C05497=1155.282,-127.548,-42.199,178.609,5.885,149.463
C05498=1155.288,-127.798,-42.191,178.606,5.885,149.464
C05499=1155.293,-128.048,-42.183,178.605,5.885,149.465
C05500=1154.872,-128.059,-42.224,178.601,5.888,149.466
C05501=1154.867,-127.809,-42.233,178.603,5.888,149.466
C05502=1154.861,-127.559,-42.241,178.605,5.888,149.465
C05503=1154.855,-127.309,-42.250,178.607,5.889,149.465
C05504=1154.850,-127.060,-42.259,178.609,5.889,149.464
C05505=1154.845,-126.809,-42.267,178.611,5.890,149.464
C05506=1154.840,-126.560,-42.275,178.613,5.890,149.463
C05507=1154.834,-126.310,-42.283,178.615,5.890,149.463
C05508=1154.829,-126.060,-42.292,178.617,5.890,149.462
C05509=1154.823,-125.811,-42.301,178.619,5.891,149.462
C05510=1154.818,-125.560,-42.309,178.621,5.891,149.461
C05511=1154.813,-125.311,-42.318,178.623,5.891,149.461
C05512=1154.807,-125.061,-42.326,178.624,5.891,149.460
C05513=1154.802,-124.811,-42.334,178.627,5.892,149.460
C05514=1154.797,-124.561,-42.343,178.628,5.892,149.459
C05515=1154.791,-124.312,-42.351,178.631,5.892,149.458
C05516=1154.786,-124.062,-42.359,178.632,5.892,149.458
C05517=1154.781,-123.812,-42.368,178.635,5.893,149.457
C05518=1154.775,-123.563,-42.377,178.636,5.893,149.457
C05519=1154.769,-123.312,-42.385,178.638,5.894,149.457
C05520=1154.764,-123.062,-42.394,178.640,5.894,149.456
C05521=1154.758,-122.813,-42.402,178.642,5.895,149.456
C05522=1154.753,-122.563,-42.411,178.644,5.894,149.455
C05523=1154.749,-122.313,-42.419,178.647,5.895,149.454
C05524=1154.743,-122.064,-42.427,178.648,5.895,149.454
C05525=1154.738,-121.814,-42.436,178.650,5.896,149.453
C05526=1154.732,-121.564,-42.445,178.652,5.896,149.453
C05527=1154.727,-121.314,-42.453,178.654,5.896,149.452
C05528=1154.721,-121.065,-42.462,178.657,5.897,149.452
C05529=1154.716,-120.815,-42.471,178.658,5.897,149.451
C05530=1154.711,-120.564,-42.479,178.661,5.897,149.451
C05531=1154.705,-120.315,-42.488,178.662,5.897,149.450
C05532=1154.700,-120.065,-42.496,178.664,5.898,149.450
C05533=1154.694,-119.816,-42.505,178.666,5.898,149.449
C05534=1154.689,-119.565,-42.514,178.669,5.898,149.449
C05535=1154.683,-119.316,-42.522,178.670,5.898,149.448
C05536=1154.678,-119.066,-42.531,178.672,5.899,149.448
C05537=1154.673,-118.816,-42.540,178.674,5.899,149.447
C05538=1154.668,-118.566,-42.549,178.676,5.900,149.447
C05539=1154.662,-118.317,-42.557,178.678,5.899,149.446
C05540=1154.656,-118.067,-42.565,178.681,5.900,149.445
C05541=1154.651,-117.817,-42.574,178.682,5.900,149.445
C05542=1154.646,-117.567,-42.583,178.684,5.901,149.444
C05543=1154.640,-117.318,-42.592,178.686,5.901,149.444
C05544=1154.635,-117.068,-42.601,178.689,5.901,149.443
C05545=1154.630,-116.818,-42.609,178.691,5.902,149.443
C05546=1154.625,-116.568,-42.618,178.692,5.902,149.442
C05547=1154.619,-116.318,-42.627,178.695,5.903,149.442
C05548=1154.614,-116.069,-42.635,178.696,5.903,149.441
C05549=1154.608,-115.819,-42.644,178.698,5.903,149.441
C05550=1154.603,-115.569,-42.653,178.700,5.903,149.440
C05551=1154.598,-115.319,-42.662,178.703,5.904,149.440
C05552=1154.592,-115.070,-42.670,178.704,5.904,149.439
C05553=1154.587,-114.820,-42.679,178.706,5.904,149.439
C05554=1154.582,-114.570,-42.688,178.708,5.904,149.438
C05555=1154.577,-114.320,-42.696,178.711,5.905,149.437
C05556=1154.571,-114.070,-42.705,178.712,5.905,149.437
C05557=1154.566,-113.821,-42.714,178.715,5.906,149.436
C05558=1154.560,-113.571,-42.723,178.717,5.906,149.436
C05559=1154.555,-113.321,-42.732,178.719,5.906,149.435
C05560=1154.549,-113.071,-42.741,178.721,5.907,149.435
C05561=1154.544,-112.821,-42.750,178.723,5.907,149.434
C05562=1154.539,-112.571,-42.759,178.725,5.907,149.434
C05563=1154.533,-112.322,-42.767,178.726,5.907,149.433
C05564=1154.528,-112.072,-42.776,178.729,5.908,149.433
C05565=1154.523,-111.822,-42.785,178.731,5.908,149.432
C05566=1154.518,-111.573,-42.794,178.733,5.908,149.432
C05567=1154.512,-111.322,-42.804,178.735,5.909,149.431
C05568=1154.507,-111.073,-42.813,178.737,5.909,149.431
C05569=1154.501,-110.823,-42.821,178.739,5.909,149.430
C05570=1154.496,-110.574,-42.830,178.741,5.909,149.429
C05571=1154.491,-110.324,-42.839,178.743,5.910,149.429
C05572=1154.485,-110.074,-42.848,178.745,5.910,149.428
C05573=1154.480,-109.824,-42.857,178.747,5.911,149.428
C05574=1154.474,-109.574,-42.866,178.750,5.911,149.427
C05575=1154.469,-109.324,-42.875,178.751,5.911,149.427
C05576=1154.463,-109.075,-42.884,178.753,5.912,149.426
C05577=1154.458,-108.825,-42.893,178.755,5.912,149.426
C05578=1154.453,-108.575,-42.901,178.758,5.912,149.425
C05579=1154.448,-108.325,-42.910,178.759,5.912,149.425
C05580=1154.442,-108.075,-42.920,178.761,5.913,149.424
C05581=1154.437,-107.825,-42.929,178.764,5.914,149.424
C05582=1154.432,-107.575,-42.938,178.766,5.913,149.423
C05583=1154.427,-107.326,-42.947,178.768,5.914,149.422
C05584=1154.421,-107.077,-42.956,178.770,5.914,149.422
C05585=1154.415,-106.827,-42.965,178.772,5.915,149.421
C05586=1154.410,-106.577,-42.974,178.774,5.914,149.421
C05587=1154.405,-106.327,-42.983,178.776,5.915,149.420
C05588=1154.400,-106.077,-42.992,178.778,5.916,149.420
C05589=1154.395,-105.828,-43.001,178.780,5.916,149.419
C05590=1154.389,-105.577,-43.010,178.782,5.916,149.419
C05591=1154.383,-105.328,-43.019,178.784,5.916,149.418
C05592=1154.379,-105.078,-43.029,178.786,5.917,149.418
C05593=1154.373,-104.828,-43.038,178.788,5.917,149.417
C05594=1154.368,-104.578,-43.047,178.791,5.917,149.416
C05595=1154.362,-104.328,-43.056,178.793,5.918,149.416
C05596=1154.357,-104.079,-43.065,178.794,5.918,149.415
C05597=1154.351,-103.829,-43.074,178.797,5.919,149.415
C05598=1154.346,-103.580,-43.084,178.799,5.918,149.414
C05599=1154.341,-103.330,-43.093,178.801,5.919,149.414
C05600=1154.335,-103.080,-43.102,178.803,5.920,149.413
C05601=1154.330,-102.808,-43.112,178.805,5.920,149.413
C05602=1154.324,-102.536,-43.121,178.807,5.920,149.412
C05603=1154.318,-102.263,-43.132,178.810,5.921,149.411
C05604=1154.312,-101.992,-43.142,178.812,5.921,149.411
C05605=1154.307,-101.742,-43.151,178.814,5.921,149.410
C05606=1154.302,-101.492,-43.160,178.816,5.922,149.410
C05607=1154.296,-101.243,-43.170,178.818,5.922,149.409
C05608=1154.291,-100.993,-43.179,178.820,5.922,149.409
C05609=1154.286,-100.743,-43.188,178.822,5.923,149.408
C05610=1154.280,-100.493,-43.197,178.824,5.923,149.407
C05611=1154.275,-100.244,-43.207,178.827,5.924,149.407
C05612=1154.270,-99.994,-43.216,178.828,5.924,149.407
C05613=1154.264,-99.744,-43.225,178.830,5.924,149.406
C05614=1154.259,-99.495,-43.235,178.833,5.925,149.405
C05615=1154.254,-99.245,-43.244,178.835,5.925,149.405
C05616=1154.248,-98.995,-43.253,178.837,5.925,149.404
C05617=1154.243,-98.745,-43.262,178.839,5.925,149.404
C05618=1154.238,-98.496,-43.272,178.841,5.926,149.403
C05619=1154.232,-98.245,-43.281,178.843,5.927,149.403
C05620=1154.227,-97.996,-43.290,178.845,5.927,149.402
C05621=1154.221,-97.746,-43.300,178.848,5.927,149.401
C05622=1154.216,-97.496,-43.309,178.850,5.928,149.401
C05623=1154.211,-97.246,-43.318,178.851,5.928,149.400
C05624=1154.205,-96.997,-43.328,178.854,5.928,149.400
C05625=1154.200,-96.747,-43.337,178.856,5.928,149.399
C05626=1154.194,-96.497,-43.348,178.858,5.929,149.399
C05627=1154.189,-96.248,-43.356,178.860,5.929,149.398
C05628=1154.185,-95.997,-43.366,178.862,5.929,149.398
C05629=1154.179,-95.747,-43.376,178.864,5.930,149.397
C05630=1154.174,-95.498,-43.385,178.867,5.931,149.397
C05631=1154.168,-95.248,-43.395,178.869,5.930,149.396
C05632=1154.163,-94.998,-43.404,178.871,5.931,149.395
C05633=1154.157,-94.748,-43.413,178.872,5.931,149.395
C05634=1154.152,-94.499,-43.423,178.875,5.932,149.394
C05635=1154.147,-94.249,-43.432,178.877,5.932,149.394
C05636=1154.142,-93.999,-43.442,178.879,5.932,149.393
C05637=1154.136,-93.750,-43.451,178.881,5.933,149.393
C05638=1154.131,-93.500,-43.461,178.884,5.933,149.392
C05639=1154.126,-93.250,-43.470,178.885,5.933,149.392
C05640=1154.120,-93.001,-43.480,178.888,5.934,149.391
C05641=1154.115,-92.751,-43.489,178.890,5.934,149.390
C05642=1154.109,-92.501,-43.499,178.892,5.934,149.390
C05643=1154.104,-92.251,-43.508,178.894,5.935,149.389
C05644=1154.099,-92.001,-43.519,178.896,5.935,149.389
C05645=1154.094,-91.751,-43.528,178.898,5.935,149.388
C05646=1154.088,-91.502,-43.538,178.900,5.936,149.388
C05647=1154.083,-91.252,-43.547,178.902,5.936,149.387
C05648=1154.078,-91.002,-43.557,178.905,5.936,149.387
C05649=1154.072,-90.752,-43.566,178.907,5.937,149.386
C05650=1154.067,-90.503,-43.576,178.909,5.937,149.386
C05651=1154.062,-90.253,-43.585,178.911,5.938,149.385
C05652=1154.056,-90.004,-43.595,178.913,5.938,149.384
C05653=1154.052,-89.753,-43.605,178.915,5.938,149.384
C05654=1154.046,-89.503,-43.615,178.918,5.939,149.383
C05655=1154.041,-89.254,-43.624,178.920,5.939,149.383
C05656=1154.035,-89.004,-43.634,178.921,5.939,149.382
C05657=1154.030,-88.755,-43.644,178.924,5.940,149.382
C05658=1154.024,-88.505,-43.653,178.926,5.941,149.381
C05659=1154.019,-88.255,-43.663,178.928,5.941,149.381
C05660=1154.014,-88.005,-43.672,178.931,5.941,149.380
C05661=1154.009,-87.755,-43.683,178.933,5.942,149.379
C05662=1154.004,-87.506,-43.692,178.934,5.942,149.379
C05663=1153.998,-87.256,-43.702,178.937,5.942,149.378
C05664=1153.992,-87.006,-43.712,178.939,5.943,149.378
C05665=1153.987,-86.757,-43.722,178.941,5.943,149.377
C05666=1153.982,-86.507,-43.731,178.943,5.944,149.377
C05667=1153.977,-86.257,-43.741,178.946,5.944,149.376
C05668=1153.972,-86.007,-43.751,178.947,5.944,149.376
C05669=1153.966,-85.757,-43.761,178.949,5.945,149.375
C05670=1153.961,-85.508,-43.770,178.952,5.945,149.374
C05671=1153.955,-85.258,-43.781,178.954,5.945,149.374
C05672=1153.951,-85.008,-43.790,178.956,5.946,149.373
C05673=1153.945,-84.758,-43.800,178.959,5.946,149.373
C05674=1153.940,-84.509,-43.810,178.960,5.946,149.372
C05675=1153.934,-84.259,-43.819,178.962,5.947,149.372
C05676=1153.929,-84.009,-43.829,178.965,5.947,149.371
C05677=1153.924,-83.759,-43.840,178.967,5.947,149.371
C05678=1153.919,-83.510,-43.850,178.969,5.948,149.370
C05679=1153.913,-83.260,-43.859,178.972,5.948,149.369
C05680=1153.907,-83.010,-43.869,178.973,5.948,149.369
C05681=1153.903,-82.761,-43.879,178.976,5.949,149.368
C05682=1153.898,-82.511,-43.889,178.978,5.950,149.368
C05683=1153.892,-82.260,-43.899,178.980,5.950,149.367
C05684=1153.887,-82.011,-43.909,178.982,5.950,149.366
C05685=1153.881,-81.762,-43.919,178.984,5.951,149.366
C05686=1153.876,-81.511,-43.929,178.986,5.951,149.365
C05687=1153.871,-81.262,-43.938,178.989,5.951,149.365
C05688=1153.865,-81.012,-43.948,178.991,5.952,149.364
C05689=1153.860,-80.762,-43.959,178.993,5.953,149.364
C05690=1153.854,-80.513,-43.969,178.995,5.952,149.363
C05691=1153.850,-80.263,-43.979,178.997,5.953,149.363
C05692=1153.844,-80.013,-43.989,179.000,5.954,149.362
C05693=1153.838,-79.763,-43.999,179.002,5.953,149.361
C05694=1153.834,-79.513,-44.009,179.004,5.954,149.361
C05695=1153.829,-79.264,-44.019,179.006,5.955,149.360
C05696=1153.823,-79.014,-44.029,179.008,5.954,149.360
C05697=1153.817,-78.765,-44.039,179.010,5.955,149.359
C05698=1153.812,-78.514,-44.050,179.013,5.956,149.359
C05699=1153.808,-78.265,-44.059,179.015,5.956,149.358
C05700=1153.802,-78.015,-44.069,179.017,5.956,149.358
C05701=1153.796,-77.766,-44.079,179.019,5.957,149.357
C05702=1153.791,-77.515,-44.090,179.022,5.958,149.356
C05703=1153.786,-77.266,-44.099,179.023,5.958,149.356
C05704=1153.781,-77.017,-44.109,179.026,5.958,149.355
C05705=1153.775,-76.745,-44.121,179.028,5.959,149.355
C05706=1153.770,-76.474,-44.132,179.031,5.959,149.354
C05707=1153.763,-76.203,-44.143,179.033,5.960,149.354
C05708=1153.758,-75.931,-44.154,179.036,5.960,149.353
C05709=1153.752,-75.681,-44.164,179.037,5.960,149.352
C05710=1153.747,-75.431,-44.174,179.040,5.961,149.352
C05711=1153.741,-75.181,-44.184,179.042,5.961,149.351
C05712=1153.736,-74.932,-44.195,179.044,5.961,149.351
C05713=1153.731,-74.682,-44.205,179.046,5.962,149.350
C05714=1153.726,-74.432,-44.215,179.049,5.963,149.349
C05715=1153.720,-74.183,-44.225,179.051,5.963,149.349
C05716=1153.715,-73.933,-44.235,179.053,5.963,149.348
C05717=1153.710,-73.683,-44.246,179.055,5.964,149.348
C05718=1153.704,-73.434,-44.256,179.058,5.964,149.347
C05719=1153.698,-73.184,-44.266,179.060,5.965,149.347
C05720=1153.694,-72.934,-44.276,179.061,5.965,149.346
C05721=1153.689,-72.685,-44.286,179.064,5.965,149.345
C05722=1153.684,-72.434,-44.297,179.066,5.966,149.345
C05723=1153.678,-72.185,-44.308,179.069,5.966,149.344
C05724=1153.673,-71.936,-44.318,179.071,5.966,149.344
C05725=1153.668,-71.686,-44.329,179.073,5.967,149.343
C05726=1153.662,-71.436,-44.339,179.075,5.967,149.343
C05727=1153.657,-71.186,-44.349,179.077,5.967,149.342
C05728=1153.652,-70.936,-44.360,179.079,5.968,149.342
C05729=1153.646,-70.687,-44.370,179.082,5.969,149.341
C05730=1153.640,-70.437,-44.380,179.084,5.969,149.340
C05731=1153.635,-70.187,-44.391,179.086,5.969,149.340
C05732=1153.630,-69.938,-44.400,179.088,5.970,149.339
C05733=1153.625,-69.687,-44.411,179.091,5.971,149.339
C05734=1153.620,-69.438,-44.421,179.093,5.971,149.338
C05735=1153.615,-69.189,-44.432,179.095,5.971,149.338
C05736=1153.610,-68.939,-44.442,179.097,5.971,149.337
C05737=1153.604,-68.689,-44.453,179.100,5.972,149.336
C05738=1153.599,-68.439,-44.463,179.102,5.973,149.336
C05739=1153.593,-68.189,-44.473,179.104,5.972,149.335
C05740=1153.588,-67.940,-44.484,179.106,5.973,149.335
C05741=1153.583,-67.690,-44.495,179.109,5.974,149.334
C05742=1153.577,-67.441,-44.505,179.111,5.974,149.334
C05743=1153.572,-67.190,-44.516,179.113,5.974,149.333
C05744=1153.567,-66.941,-44.526,179.115,5.975,149.332
C05745=1153.562,-66.691,-44.537,179.117,5.976,149.332
C05746=1153.557,-66.442,-44.547,179.120,5.976,149.331
C05747=1153.552,-66.191,-44.558,179.122,5.977,149.331
C05748=1153.546,-65.942,-44.568,179.124,5.977,149.330
C05749=1153.540,-65.692,-44.578,179.127,5.977,149.329
C05750=1153.536,-65.443,-44.590,179.129,5.978,149.329
C05751=1153.530,-65.193,-44.600,179.131,5.979,149.329
C05752=1153.525,-64.943,-44.611,179.133,5.978,149.328
C05753=1153.520,-64.693,-44.621,179.135,5.979,149.327
C05754=1153.515,-64.444,-44.632,179.138,5.979,149.327
C05755=1153.509,-64.194,-44.642,179.140,5.980,149.326
C05756=1153.504,-63.944,-44.653,179.142,5.981,149.326
C05757=1153.498,-63.694,-44.664,179.144,5.981,149.325
C05758=1153.493,-63.445,-44.675,179.146,5.981,149.324
C05759=1153.488,-63.195,-44.685,179.149,5.982,149.324
C05760=1153.483,-62.945,-44.696,179.151,5.983,149.323
C05761=1153.477,-62.696,-44.707,179.153,5.982,149.323
C05762=1153.472,-62.446,-44.717,179.156,5.983,149.322
C05763=1153.467,-62.196,-44.727,179.158,5.984,149.322
C05764=1153.462,-61.946,-44.739,179.160,5.984,149.321
C05765=1153.456,-61.697,-44.749,179.163,5.985,149.320
C05766=1153.451,-61.447,-44.759,179.165,5.984,149.320
C05767=1153.446,-61.198,-44.770,179.167,5.985,149.319
C05768=1153.440,-60.947,-44.782,179.169,5.986,149.319
C05769=1153.435,-60.698,-44.792,179.172,5.986,149.318
C05770=1153.430,-60.448,-44.803,179.174,5.987,149.318
C05771=1153.425,-60.198,-44.813,179.176,5.987,149.317
C05772=1153.420,-59.949,-44.825,179.178,5.988,149.316
C05773=1153.414,-59.699,-44.835,179.180,5.988,149.316
C05774=1153.410,-59.450,-44.846,179.183,5.989,149.315
C05775=1153.404,-59.200,-44.856,179.185,5.990,149.315
C05776=1153.398,-58.950,-44.867,179.187,5.989,149.314
C05777=1153.394,-58.700,-44.879,179.190,5.990,149.314
C05778=1153.388,-58.450,-44.889,179.192,5.990,149.313
C05779=1153.383,-58.201,-44.900,179.194,5.991,149.312
C05780=1153.378,-57.951,-44.910,179.197,5.992,149.312
C05781=1153.373,-57.702,-44.922,179.199,5.992,149.311
C05782=1153.367,-57.452,-44.933,179.201,5.992,149.311
C05783=1153.362,-57.202,-44.944,179.204,5.993,149.310
C05784=1153.357,-56.952,-44.954,179.206,5.993,149.310
C05785=1153.352,-56.703,-44.965,179.208,5.994,149.309
C05786=1153.347,-56.453,-44.976,179.210,5.994,149.308
C05787=1153.341,-56.203,-44.987,179.212,5.995,149.308
C05788=1153.336,-55.953,-44.998,179.215,5.995,149.307
C05789=1153.331,-55.704,-45.009,179.217,5.996,149.307
C05790=1153.325,-55.454,-45.019,179.220,5.996,149.306
C05791=1153.320,-55.204,-45.031,179.222,5.997,149.306
C05792=1153.314,-54.955,-45.042,179.223,5.997,149.305
C05793=1153.310,-54.705,-45.053,179.226,5.997,149.304
C05794=1153.305,-54.455,-45.063,179.228,5.998,149.304
C05795=1153.299,-54.205,-45.075,179.231,5.999,149.303
C05796=1153.294,-53.956,-45.086,179.233,5.999,149.303
C05797=1153.288,-53.706,-45.096,179.235,5.999,149.302
C05798=1153.284,-53.457,-45.108,179.237,6.000,149.301
C05799=1153.278,-53.206,-45.119,179.240,6.001,149.301
C05800=1153.273,-52.957,-45.130,179.242,6.001,149.300
C05801=1153.268,-52.708,-45.141,179.244,6.002,149.300
C05802=1153.262,-52.457,-45.152,179.247,6.002,149.299
C05803=1153.257,-52.208,-45.163,179.249,6.002,149.299
C05804=1153.252,-51.958,-45.175,179.251,6.003,149.298
C05805=1153.247,-51.708,-45.185,179.254,6.003,149.297
C05806=1153.241,-51.459,-45.197,179.256,6.004,149.297
C05807=1153.236,-51.209,-45.208,179.258,6.005,149.296
C05808=1153.231,-50.959,-45.218,179.261,6.005,149.296
C05809=1153.225,-50.689,-45.230,179.263,6.006,149.295
C05810=1153.220,-50.418,-45.243,179.266,6.006,149.294
C05811=1153.214,-50.148,-45.255,179.268,6.007,149.294
C05812=1153.208,-49.877,-45.267,179.271,6.007,149.293
C05813=1153.203,-49.627,-45.278,179.273,6.008,149.293
C05814=1153.197,-49.378,-45.290,179.275,6.008,149.292
C05815=1153.192,-49.128,-45.301,179.277,6.008,149.292
C05816=1153.187,-48.878,-45.311,179.280,6.009,149.291
C05817=1153.182,-48.628,-45.323,179.282,6.010,149.290
C05818=1153.177,-48.379,-45.334,179.285,6.010,149.290
C05819=1153.172,-48.129,-45.346,179.287,6.011,149.289
C05820=1153.166,-47.879,-45.357,179.289,6.012,149.289
C05821=1153.161,-47.630,-45.368,179.291,6.011,149.288
C05822=1153.155,-47.380,-45.379,179.293,6.012,149.288
C05823=1153.151,-47.130,-45.391,179.296,6.012,149.287
C05824=1153.145,-46.881,-45.402,179.298,6.013,149.286
C05825=1153.140,-46.631,-45.413,179.301,6.014,149.286
C05826=1153.135,-46.381,-45.424,179.303,6.014,149.285
C05827=1153.130,-46.131,-45.436,179.306,6.015,149.284
C05828=1153.124,-45.882,-45.447,179.307,6.015,149.284
C05829=1153.119,-45.632,-45.459,179.310,6.016,149.284
C05830=1153.114,-45.383,-45.470,179.312,6.016,149.283
C05831=1153.108,-45.132,-45.481,179.314,6.017,149.282
C05832=1153.103,-44.883,-45.492,179.317,6.017,149.282
C05833=1153.098,-44.633,-45.504,179.319,6.018,149.281
C05834=1153.093,-44.384,-45.515,179.322,6.018,149.280
C05835=1153.088,-44.134,-45.527,179.324,6.019,149.280
C05836=1153.082,-43.885,-45.538,179.327,6.020,149.279
C05837=1153.077,-43.635,-45.550,179.328,6.020,149.279
C05838=1153.072,-43.385,-45.561,179.331,6.020,149.278
C05839=1153.066,-43.135,-45.573,179.333,6.021,149.278
C05840=1153.061,-42.886,-45.583,179.335,6.022,149.277
C05841=1153.056,-42.636,-45.595,179.338,6.022,149.276
C05842=1153.051,-42.386,-45.607,179.340,6.023,149.276
C05843=1153.046,-42.136,-45.619,179.343,6.023,149.275
C05844=1153.041,-41.887,-45.630,179.345,6.024,149.275
C05845=1153.035,-41.637,-45.641,179.348,6.024,149.274
C05846=1153.030,-41.388,-45.653,179.349,6.024,149.274
C05847=1153.025,-41.138,-45.665,179.352,6.025,149.273
C05848=1153.020,-40.888,-45.676,179.354,6.026,149.272
C05849=1153.015,-40.638,-45.688,179.356,6.026,149.272
C05850=1153.010,-40.389,-45.699,179.359,6.027,149.271
C05851=1153.004,-40.140,-45.711,179.361,6.028,149.271
C05852=1152.999,-39.890,-45.722,179.364,6.028,149.270
C05853=1152.994,-39.640,-45.734,179.366,6.029,149.270
C05854=1152.988,-39.390,-45.746,179.369,6.029,149.269
C05855=1152.984,-39.140,-45.757,179.371,6.030,149.268
C05856=1152.978,-38.891,-45.768,179.373,6.030,149.268
C05857=1152.972,-38.641,-45.780,179.375,6.030,149.267
C05858=1152.968,-38.392,-45.792,179.378,6.031,149.267
C05859=1152.962,-38.142,-45.803,179.380,6.032,149.266
C05860=1152.957,-37.892,-45.815,179.382,6.032,149.266
C05861=1152.952,-37.642,-45.827,179.385,6.033,149.265
C05862=1152.947,-37.392,-45.839,179.387,6.034,149.264
C05863=1152.942,-37.144,-45.850,179.390,6.034,149.264
C05864=1152.936,-36.894,-45.862,179.392,6.035,149.263
C05865=1152.931,-36.644,-45.874,179.395,6.035,149.263
C05866=1152.926,-36.394,-45.885,179.397,6.036,149.262
C05867=1152.921,-36.144,-45.897,179.399,6.036,149.261
C05868=1152.915,-35.894,-45.909,179.401,6.036,149.261
C05869=1152.910,-35.645,-45.920,179.404,6.037,149.260
C05870=1152.905,-35.395,-45.932,179.406,6.038,149.260
C05871=1152.899,-35.146,-45.944,179.409,6.038,149.259
C05872=1152.895,-34.897,-45.956,179.411,6.039,149.259
C05873=1152.889,-34.647,-45.968,179.413,6.040,149.258
C05874=1152.884,-34.397,-45.979,179.416,6.040,149.257
C05875=1152.878,-34.147,-45.991,179.418,6.041,149.257
C05876=1152.874,-33.897,-46.003,179.420,6.041,149.256
C05877=1152.869,-33.648,-46.015,179.423,6.042,149.256
C05878=1152.863,-33.398,-46.027,179.425,6.042,149.255
C05879=1152.858,-33.148,-46.038,179.427,6.043,149.255
C05880=1152.853,-32.898,-46.050,179.430,6.044,149.254
C05881=1152.848,-32.648,-46.062,179.432,6.044,149.253
C05882=1152.842,-32.399,-46.075,179.435,6.045,149.253
C05883=1152.837,-32.150,-46.086,179.437,6.046,149.252
C05884=1152.832,-31.900,-46.098,179.439,6.045,149.252
C05885=1152.827,-31.651,-46.110,179.441,6.046,149.251
C05886=1152.821,-31.401,-46.122,179.444,6.047,149.250
C05887=1152.816,-31.151,-46.133,179.446,6.047,149.250
C05888=1152.811,-30.901,-46.145,179.448,6.048,149.249
C05889=1152.806,-30.652,-46.158,179.451,6.049,149.249
C05890=1152.800,-30.402,-46.170,179.453,6.049,149.248
C05891=1152.795,-30.152,-46.182,179.456,6.050,149.248
C05892=1152.791,-29.903,-46.194,179.458,6.051,149.247
C05893=1152.785,-29.653,-46.206,179.461,6.051,149.246
C05894=1152.780,-29.403,-46.217,179.463,6.052,149.246
C05895=1152.775,-29.154,-46.230,179.466,6.052,149.245
C05896=1152.769,-28.904,-46.242,179.468,6.053,149.245
C05897=1152.765,-28.655,-46.253,179.470,6.053,149.244
C05898=1152.759,-28.405,-46.266,179.473,6.054,149.244
C05899=1152.754,-28.155,-46.278,179.475,6.055,149.243
C05900=1152.749,-27.905,-46.290,179.477,6.055,149.242
C05901=1152.743,-27.656,-46.302,179.480,6.056,149.242
C05902=1152.738,-27.406,-46.314,179.482,6.057,149.241
C05903=1152.734,-27.157,-46.326,179.485,6.057,149.241
C05904=1152.728,-26.907,-46.338,179.487,6.058,149.240
C05905=1152.723,-26.657,-46.350,179.489,6.059,149.240
C05906=1152.718,-26.408,-46.362,179.492,6.059,149.239
C05907=1152.712,-26.158,-46.374,179.494,6.060,149.238
C05908=1152.707,-25.909,-46.387,179.497,6.060,149.238
C05909=1152.702,-25.659,-46.399,179.499,6.061,149.237
C05910=1152.697,-25.409,-46.411,179.502,6.062,149.237
C05911=1152.691,-25.159,-46.423,179.504,6.062,149.236
C05912=1152.687,-24.910,-46.435,179.507,6.063,149.235
C05913=1152.681,-24.640,-46.449,179.509,6.064,149.235
C05914=1152.675,-24.369,-46.462,179.511,6.064,149.234
C05915=1152.670,-24.100,-46.475,179.514,6.064,149.234
C05916=1152.664,-23.830,-46.488,179.517,6.065,149.233
C05917=1152.659,-23.581,-46.501,179.519,6.066,149.232
C05918=1152.654,-23.331,-46.513,179.521,6.066,149.232
C05919=1152.649,-23.081,-46.525,179.524,6.067,149.231
C05920=1152.643,-22.832,-46.537,179.526,6.068,149.231
C05921=1152.638,-22.582,-46.550,179.529,6.068,149.230
C05922=1152.633,-22.332,-46.562,179.531,6.069,149.230
C05923=1152.628,-22.082,-46.574,179.533,6.069,149.229
C05924=1152.623,-21.832,-46.586,179.536,6.070,149.228
C05925=1152.618,-21.583,-46.599,179.538,6.071,149.228
C05926=1152.613,-21.334,-46.612,179.540,6.071,149.227
C05927=1152.607,-21.084,-46.623,179.543,6.072,149.227
C05928=1152.602,-20.834,-46.636,179.545,6.073,149.226
C05929=1152.597,-20.585,-46.648,179.548,6.073,149.225
C05930=1152.592,-20.335,-46.661,179.550,6.074,149.225
C05931=1152.586,-20.086,-46.673,179.553,6.074,149.224
C05932=1152.582,-19.835,-46.685,179.555,6.075,149.224
C05933=1152.576,-19.586,-46.698,179.558,6.075,149.223
C05934=1152.571,-19.337,-46.711,179.560,6.076,149.223
C05935=1152.566,-19.087,-46.722,179.562,6.077,149.222
C05936=1152.561,-18.837,-46.735,179.565,6.077,149.221
C05937=1152.555,-18.588,-46.748,179.567,6.078,149.221
C05938=1152.549,-18.338,-46.760,179.569,6.079,149.220
C05939=1152.545,-18.088,-46.773,179.572,6.080,149.220
C05940=1152.540,-17.838,-46.786,179.575,6.081,149.219
C05941=1152.534,-17.588,-46.798,179.577,6.082,149.219
C05942=1152.529,-17.339,-46.810,179.580,6.082,149.218
C05943=1152.524,-17.090,-46.823,179.582,6.083,149.217
C05944=1152.519,-16.841,-46.835,179.585,6.083,149.217
C05945=1152.514,-16.590,-46.848,179.587,6.084,149.216
C05946=1152.509,-16.341,-46.860,179.589,6.084,149.216
C05947=1152.504,-16.091,-46.873,179.592,6.085,149.215
C05948=1152.498,-15.842,-46.886,179.594,6.086,149.214
C05949=1152.493,-15.592,-46.898,179.596,6.086,149.214
C05950=1152.488,-15.342,-46.911,179.599,6.087,149.213
C05951=1152.483,-15.092,-46.924,179.601,6.088,149.213
C05952=1152.478,-14.843,-46.936,179.604,6.088,149.212
C05953=1152.473,-14.594,-46.949,179.606,6.089,149.212
C05954=1152.468,-14.344,-46.961,179.609,6.089,149.211
C05955=1152.462,-14.093,-46.974,179.611,6.090,149.210
C05956=1152.457,-13.844,-46.987,179.614,6.091,149.210
C05957=1152.452,-13.595,-46.999,179.616,6.091,149.209
C05958=1152.447,-13.346,-47.012,179.618,6.092,149.209
C05959=1152.442,-13.096,-47.025,179.621,6.093,149.208
C05960=1152.437,-12.846,-47.038,179.623,6.093,149.207
C05961=1152.431,-12.596,-47.050,179.625,6.094,149.207
C05962=1152.426,-12.347,-47.063,179.629,6.095,149.206
C05963=1152.421,-12.097,-47.075,179.631,6.096,149.206
C05964=1152.416,-11.847,-47.088,179.634,6.096,149.205
C05965=1152.411,-11.598,-47.101,179.636,6.097,149.205
C05966=1152.405,-11.348,-47.114,179.638,6.098,149.204
C05967=1152.400,-11.099,-47.127,179.641,6.098,149.203
C05968=1152.395,-10.849,-47.140,179.643,6.099,149.203
C05969=1152.390,-10.600,-47.152,179.645,6.100,149.202
C05970=1152.384,-10.350,-47.165,179.648,6.100,149.202
C05971=1152.380,-10.100,-47.178,179.650,6.101,149.201
C05972=1152.375,-9.851,-47.191,179.652,6.102,149.201
C05973=1152.370,-9.601,-47.204,179.655,6.102,149.200
C05974=1152.364,-9.352,-47.217,179.657,6.103,149.200
C05975=1152.359,-9.102,-47.230,179.660,6.103,149.199
C05976=1152.354,-8.852,-47.242,179.663,6.105,149.198
C05977=1152.348,-8.603,-47.255,179.665,6.105,149.198
C05978=1152.344,-8.353,-47.268,179.668,6.106,149.197
C05979=1152.339,-8.103,-47.281,179.670,6.107,149.197
C05980=1152.334,-7.854,-47.294,179.672,6.107,149.196
C05981=1152.328,-7.604,-47.307,179.675,6.108,149.195
C05982=1152.323,-7.355,-47.320,179.677,6.109,149.195
C05983=1152.318,-7.105,-47.332,179.680,6.109,149.194
C05984=1152.313,-6.855,-47.346,179.682,6.110,149.194
C05985=1152.308,-6.606,-47.359,179.685,6.110,149.193
C05986=1152.303,-6.356,-47.371,179.687,6.111,149.193
C05987=1152.297,-6.106,-47.385,179.690,6.112,149.192
C05988=1152.292,-5.857,-47.397,179.692,6.113,149.191
C05989=1152.287,-5.608,-47.411,179.695,6.114,149.191
C05990=1152.282,-5.358,-47.424,179.697,6.114,149.190
C05991=1152.277,-5.108,-47.437,179.700,6.115,149.190
C05992=1152.271,-4.859,-47.450,179.702,6.116,149.189
C05993=1152.267,-4.609,-47.463,179.705,6.116,149.188
C05994=1152.261,-4.359,-47.476,179.707,6.117,149.188
C05995=1152.256,-4.109,-47.489,179.709,6.118,149.188
C05996=1152.251,-3.860,-47.502,179.712,6.119,149.187
C05997=1152.246,-3.611,-47.516,179.714,6.120,149.186
C05998=1152.241,-3.361,-47.529,179.717,6.120,149.186
C05999=1152.236,-3.111,-47.541,179.719,6.121,149.185
C06000=1152.231,-2.861,-47.555,179.722,6.122,149.185
C06001=1152.226,-2.612,-47.568,179.724,6.122,149.184
C06002=1152.220,-2.363,-47.581,179.727,6.123,149.183
C06003=1152.215,-2.113,-47.594,179.729,6.124,149.183
C06004=1152.210,-1.863,-47.607,179.732,6.124,149.182
C06005=1152.205,-1.614,-47.621,179.734,6.126,149.182
C06006=1152.199,-1.364,-47.634,179.737,6.126,149.181
C06007=1152.194,-1.115,-47.647,179.739,6.127,149.181
C06008=1152.190,-0.865,-47.660,179.742,6.127,149.180
C06009=1152.184,-0.616,-47.674,179.744,6.128,149.179
C06010=1152.180,-0.366,-47.687,179.747,6.129,149.179
C06011=1152.174,-0.116,-47.700,179.749,6.129,149.178
C06012=1152.169,0.134,-47.713,179.752,6.131,149.178
C06013=1152.164,0.383,-47.727,179.754,6.131,149.177
C06014=1152.159,0.632,-47.739,179.757,6.132,149.176
C06015=1152.153,0.883,-47.753,179.759,6.133,149.176
C06016=1152.148,1.132,-47.767,179.762,6.133,149.175
C06017=1152.143,1.401,-47.781,179.764,6.134,149.175
C06018=1152.137,1.671,-47.796,179.767,6.135,149.174
C06019=1152.132,1.941,-47.810,179.770,6.136,149.173
C06020=1152.126,2.209,-47.824,179.772,6.136,149.173
C06021=1152.121,2.460,-47.837,179.775,6.138,149.172
C06022=1152.116,2.709,-47.851,179.777,6.139,149.172
C06023=1152.111,2.959,-47.864,179.780,6.139,149.171
C06024=1152.106,3.208,-47.878,179.782,6.140,149.171
C06025=1152.101,3.458,-47.891,179.785,6.140,149.170
C06026=1152.095,3.707,-47.904,179.787,6.141,149.170
C06027=1152.091,3.957,-47.918,179.790,6.142,149.169
C06028=1152.085,4.206,-47.931,179.792,6.143,149.168
C06029=1152.080,4.456,-47.946,179.795,6.144,149.168
C06030=1152.075,4.705,-47.958,179.797,6.144,149.167
C06031=1152.070,4.955,-47.972,179.800,6.145,149.167
C06032=1152.065,5.204,-47.985,179.802,6.146,149.166
C06033=1152.060,5.454,-47.999,179.805,6.146,149.165
C06034=1152.054,5.704,-48.013,179.808,6.148,149.165
C06035=1152.050,5.953,-48.026,179.810,6.148,149.164
C06036=1152.044,6.203,-48.039,179.812,6.149,149.164
C06037=1152.039,6.452,-48.054,179.815,6.150,149.163
C06038=1152.035,6.703,-48.067,179.817,6.150,149.163
C06039=1152.029,6.952,-48.081,179.820,6.152,149.162
C06040=1152.024,7.202,-48.094,179.823,6.152,149.161
C06041=1152.019,7.451,-48.107,179.825,6.153,149.161
C06042=1152.014,7.700,-48.122,179.827,6.154,149.160
C06043=1152.008,7.950,-48.135,179.830,6.154,149.160
C06044=1152.004,8.199,-48.149,179.832,6.155,149.159
C06045=1151.999,8.450,-48.162,179.835,6.156,149.159
C06046=1151.993,8.699,-48.176,179.838,6.157,149.158
C06047=1151.989,8.948,-48.190,179.840,6.158,149.158
C06048=1151.983,9.198,-48.203,179.843,6.158,149.157
C06049=1151.978,9.447,-48.217,179.845,6.159,149.156
C06050=1151.973,9.698,-48.231,179.848,6.160,149.156
C06051=1151.968,9.946,-48.244,179.850,6.161,149.155
C06052=1151.963,10.196,-48.258,179.853,6.162,149.155
C06053=1151.957,10.446,-48.272,179.855,6.162,149.154
C06054=1151.952,10.695,-48.286,179.858,6.163,149.153
C06055=1151.948,10.945,-48.300,179.860,6.164,149.153
C06056=1151.942,11.194,-48.313,179.863,6.165,149.152
C06057=1151.937,11.444,-48.327,179.865,6.166,149.152
C06058=1151.932,11.693,-48.341,179.867,6.167,149.151
C06059=1151.927,11.943,-48.355,179.870,6.167,149.151
C06060=1151.922,12.193,-48.368,179.873,6.169,149.150
C06061=1151.917,12.442,-48.382,179.875,6.169,149.150
C06062=1151.912,12.692,-48.396,179.878,6.170,149.149
C06063=1151.906,12.942,-48.410,179.880,6.170,149.148
C06064=1151.901,13.191,-48.424,179.882,6.171,149.148
C06065=1151.897,13.440,-48.438,179.886,6.172,149.147
C06066=1151.892,13.690,-48.452,179.888,6.173,149.147
C06067=1151.886,13.939,-48.466,179.890,6.174,149.146
C06068=1151.881,14.189,-48.479,179.893,6.174,149.146
C06069=1151.876,14.439,-48.494,179.896,6.176,149.145
C06070=1151.870,14.688,-48.507,179.898,6.177,149.145
C06071=1151.866,14.938,-48.521,179.901,6.177,149.144
C06072=1151.861,15.187,-48.535,179.903,6.178,149.143
C06073=1151.855,15.437,-48.549,179.906,6.179,149.143
C06074=1151.850,15.687,-48.563,179.908,6.180,149.142
C06075=1151.845,15.936,-48.577,179.910,6.181,149.142
C06076=1151.840,16.186,-48.591,179.913,6.181,149.141
C06077=1151.835,16.435,-48.605,179.915,6.182,149.141
C06078=1151.830,16.685,-48.620,179.919,6.183,149.140
C06079=1151.825,16.934,-48.634,179.921,6.184,149.140
C06080=1151.819,17.183,-48.648,179.923,6.185,149.139
C06081=1151.815,17.433,-48.661,179.926,6.185,149.138
C06082=1151.810,17.683,-48.675,179.929,6.187,149.138
C06083=1151.805,17.933,-48.689,179.931,6.187,149.137
C06084=1151.799,18.182,-48.703,179.934,6.188,149.137
C06085=1151.794,18.432,-48.718,179.936,6.189,149.136
C06086=1151.789,18.681,-48.732,179.939,6.190,149.135
C06087=1151.784,18.931,-48.746,179.941,6.191,149.135
C06088=1151.779,19.180,-48.760,179.944,6.191,149.134
C06089=1151.774,19.430,-48.774,179.946,6.192,149.134
C06090=1151.769,19.679,-48.789,179.949,6.193,149.133
C06091=1151.764,19.929,-48.803,179.951,6.194,149.133
C06092=1151.758,20.178,-48.817,179.954,6.195,149.132
C06093=1151.754,20.428,-48.831,179.957,6.196,149.132
C06094=1151.749,20.678,-48.845,179.959,6.197,149.131
C06095=1151.744,20.927,-48.860,179.962,6.198,149.130
C06096=1151.739,21.177,-48.874,179.964,6.198,149.130
C06097=1151.733,21.426,-48.888,179.967,6.200,149.129
C06098=1151.728,21.676,-48.902,179.969,6.200,149.129
C06099=1151.723,21.925,-48.916,179.972,6.201,149.128
C06100=1151.718,22.175,-48.931,179.974,6.202,149.128
C06101=1151.714,22.424,-48.946,179.977,6.203,149.127
C06102=1151.708,22.673,-48.959,179.979,6.204,149.127
C06103=1151.703,22.923,-48.974,179.982,6.204,149.126
C06104=1151.698,23.173,-48.988,179.985,6.206,149.125
C06105=1151.693,23.422,-49.002,179.987,6.207,149.125
C06106=1151.687,23.672,-49.017,179.990,6.207,149.124
C06107=1151.683,23.922,-49.031,179.992,6.208,149.124
C06108=1151.677,24.171,-49.045,179.995,6.209,149.123
C06109=1151.672,24.420,-49.060,179.997,6.210,149.123
C06110=1151.667,24.670,-49.075,180.000,6.211,149.122
C06111=1151.662,24.920,-49.089,-179.997,6.212,149.122
C06112=1151.657,25.169,-49.103,-179.995,6.213,149.121
C06113=1151.653,25.419,-49.117,-179.993,6.214,149.120
C06114=1151.647,25.668,-49.131,-179.990,6.214,149.120
C06115=1151.642,25.917,-49.147,-179.987,6.216,149.119
C06116=1151.637,26.167,-49.161,-179.984,6.216,149.119
C06117=1151.632,26.417,-49.176,-179.982,6.217,149.118
C06118=1151.627,26.667,-49.190,-179.980,6.219,149.118
C06119=1151.622,26.916,-49.205,-179.977,6.219,149.117
C06120=1151.617,27.165,-49.219,-179.975,6.220,149.117
C06121=1151.611,27.435,-49.235,-179.971,6.221,149.116
C06122=1151.606,27.704,-49.250,-179.969,6.222,149.115
C06123=1151.600,27.972,-49.266,-179.966,6.223,149.115
C06124=1151.595,28.241,-49.281,-179.963,6.224,149.114
C06125=1151.589,28.491,-49.296,-179.961,6.225,149.114
C06126=1151.585,28.740,-49.311,-179.958,6.226,149.113
C06127=1151.580,28.990,-49.326,-179.956,6.227,149.112
C06128=1151.575,29.239,-49.340,-179.953,6.228,149.112
C06129=1151.569,29.489,-49.355,-179.950,6.229,149.111
C06130=1151.564,29.738,-49.370,-179.948,6.229,149.111
C06131=1151.559,29.988,-49.384,-179.946,6.230,149.110
C06132=1151.555,30.237,-49.399,-179.942,6.231,149.110
C06133=1151.550,30.487,-49.413,-179.940,6.232,149.109
C06134=1151.544,30.736,-49.429,-179.938,6.233,149.109
C06135=1151.539,30.986,-49.443,-179.935,6.234,149.108
C06136=1151.535,31.236,-49.457,-179.933,6.235,149.108
C06137=1151.529,31.485,-49.473,-179.930,6.235,149.107
C06138=1151.524,31.735,-49.487,-179.927,6.237,149.106
C06139=1151.520,31.984,-49.502,-179.925,6.238,149.106
C06140=1151.514,32.233,-49.516,-179.922,6.238,149.105
C06141=1151.509,32.482,-49.532,-179.919,6.240,149.105
C06142=1151.504,32.732,-49.546,-179.917,6.241,149.104
C06143=1151.499,32.982,-49.560,-179.914,6.242,149.104
C06144=1151.493,33.231,-49.576,-179.912,6.243,149.103
C06145=1151.488,33.481,-49.590,-179.909,6.243,149.103
C06146=1151.484,33.730,-49.605,-179.906,6.245,149.102
C06147=1151.478,33.980,-49.620,-179.904,6.246,149.101
C06148=1151.473,34.229,-49.635,-179.901,6.246,149.101
C06149=1151.468,34.479,-49.649,-179.899,6.248,149.100
C06150=1151.463,34.728,-49.665,-179.896,6.248,149.100
C06151=1151.459,34.978,-49.680,-179.894,6.249,149.099
C06152=1151.453,35.228,-49.695,-179.891,6.251,149.099
C06153=1151.449,35.477,-49.710,-179.888,6.251,149.098
C06154=1151.444,35.727,-49.724,-179.886,6.252,149.098
C06155=1151.438,35.976,-49.740,-179.883,6.253,149.097
C06156=1151.433,36.226,-49.754,-179.881,6.254,149.096
C06157=1151.428,36.475,-49.770,-179.878,6.255,149.096
C06158=1151.423,36.724,-49.785,-179.875,6.256,149.095
C06159=1151.418,36.974,-49.799,-179.873,6.257,149.095
C06160=1151.413,37.224,-49.815,-179.870,6.258,149.094
C06161=1151.408,37.473,-49.829,-179.868,6.259,149.094
C06162=1151.403,37.723,-49.845,-179.865,6.260,149.093
C06163=1151.398,37.972,-49.860,-179.863,6.261,149.093
C06164=1151.392,38.222,-49.874,-179.860,6.262,149.092
C06165=1151.388,38.471,-49.889,-179.857,6.263,149.092
C06166=1151.382,38.720,-49.905,-179.854,6.264,149.091
C06167=1151.377,38.970,-49.919,-179.852,6.265,149.090
C06168=1151.373,39.219,-49.934,-179.850,6.266,149.090
C06169=1151.368,39.469,-49.950,-179.847,6.267,149.089
C06170=1151.363,39.718,-49.965,-179.845,6.268,149.089
C06171=1151.357,39.968,-49.980,-179.842,6.269,149.088
C06172=1151.353,40.217,-49.995,-179.839,6.270,149.088
C06173=1151.347,40.467,-50.011,-179.836,6.271,149.087
C06174=1151.342,40.716,-50.026,-179.834,6.272,149.087
C06175=1151.337,40.966,-50.041,-179.832,6.273,149.086
C06176=1151.332,41.215,-50.056,-179.829,6.274,149.085
C06177=1151.328,41.465,-50.071,-179.826,6.275,149.085
C06178=1151.322,41.715,-50.087,-179.823,6.276,149.084
C06179=1151.317,41.964,-50.101,-179.821,6.277,149.084
C06180=1151.312,42.214,-50.117,-179.818,6.277,149.083
C06181=1151.307,42.463,-50.132,-179.816,6.279,149.083
C06182=1151.302,42.712,-50.148,-179.813,6.280,149.082
C06183=1151.297,42.961,-50.163,-179.810,6.281,149.082
C06184=1151.292,43.211,-50.178,-179.808,6.282,149.081
C06185=1151.287,43.461,-50.193,-179.805,6.283,149.081
C06186=1151.282,43.710,-50.208,-179.803,6.284,149.080
C06187=1151.277,43.960,-50.224,-179.800,6.285,149.079
C06188=1151.272,44.209,-50.239,-179.797,6.286,149.079
C06189=1151.267,44.458,-50.255,-179.795,6.287,149.079
C06190=1151.262,44.708,-50.270,-179.792,6.288,149.078
C06191=1151.257,44.958,-50.285,-179.790,6.289,149.077
C06192=1151.252,45.207,-50.301,-179.786,6.290,149.077
C06193=1151.246,45.456,-50.317,-179.784,6.291,149.076
C06194=1151.242,45.706,-50.332,-179.782,6.292,149.076
C06195=1151.237,45.956,-50.348,-179.779,6.293,149.075
C06196=1151.232,46.205,-50.363,-179.777,6.294,149.075
C06197=1151.227,46.454,-50.378,-179.774,6.296,149.074
C06198=1151.222,46.703,-50.394,-179.771,6.296,149.074
C06199=1151.217,46.954,-50.410,-179.768,6.298,149.073
C06200=1151.212,47.203,-50.425,-179.766,6.299,149.073
C06201=1151.207,47.452,-50.440,-179.764,6.299,149.072
C06202=1151.201,47.701,-50.456,-179.761,6.301,149.071
C06203=1151.197,47.951,-50.471,-179.758,6.302,149.071
C06204=1151.192,48.201,-50.487,-179.755,6.303,149.070
C06205=1151.187,48.450,-50.502,-179.753,6.304,149.070
C06206=1151.182,48.699,-50.517,-179.750,6.305,149.069
C06207=1151.177,48.949,-50.533,-179.748,6.306,149.069
C06208=1151.172,49.199,-50.549,-179.745,6.307,149.068
C06209=1151.166,49.448,-50.565,-179.742,6.308,149.068
C06210=1151.162,49.697,-50.580,-179.740,6.309,149.067
C06211=1151.157,49.947,-50.595,-179.737,6.310,149.067
C06212=1151.152,50.197,-50.611,-179.735,6.311,149.066
C06213=1151.146,50.446,-50.627,-179.732,6.313,149.066
C06214=1151.142,50.695,-50.643,-179.729,6.313,149.065
C06215=1151.137,50.945,-50.658,-179.727,6.315,149.065
C06216=1151.132,51.194,-50.674,-179.724,6.316,149.064
C06217=1151.127,51.444,-50.690,-179.721,6.317,149.063
C06218=1151.121,51.694,-50.705,-179.719,6.318,149.063
C06219=1151.117,51.943,-50.720,-179.716,6.319,149.062
C06220=1151.112,52.192,-50.737,-179.714,6.320,149.062
C06221=1151.107,52.442,-50.753,-179.711,6.321,149.061
C06222=1151.102,52.691,-50.768,-179.708,6.322,149.061
C06223=1151.097,52.941,-50.784,-179.705,6.324,149.060
C06224=1151.091,53.190,-50.800,-179.703,6.324,149.060
C06225=1151.086,53.459,-50.817,-179.700,6.326,149.059
C06226=1151.081,53.727,-50.833,-179.697,6.326,149.059
C06227=1151.075,53.996,-50.850,-179.695,6.328,149.058
C06228=1151.071,54.265,-50.868,-179.691,6.329,149.057
C06229=1151.065,54.514,-50.884,-179.689,6.330,149.057
C06230=1151.060,54.763,-50.900,-179.686,6.331,149.056
C06231=1151.055,55.013,-50.915,-179.684,6.332,149.056
C06232=1151.050,55.262,-50.932,-179.681,6.333,149.055
C06233=1151.045,55.512,-50.948,-179.679,6.334,149.055
C06234=1151.040,55.761,-50.963,-179.676,6.336,149.054
C06235=1151.035,56.010,-50.980,-179.673,6.336,149.054
C06236=1151.030,56.260,-50.996,-179.670,6.338,149.053
C06237=1151.025,56.510,-51.011,-179.668,6.339,149.053
C06238=1151.020,56.758,-51.027,-179.665,6.340,149.052
C06239=1151.016,57.008,-51.043,-179.663,6.341,149.052
C06240=1151.010,57.258,-51.058,-179.660,6.342,149.051
C06241=1151.006,57.507,-51.075,-179.657,6.343,149.051
C06242=1151.000,57.756,-51.091,-179.655,6.345,149.050
C06243=1150.996,58.006,-51.107,-179.652,6.345,149.049
C06244=1150.991,58.255,-51.123,-179.649,6.347,149.049
C06245=1150.985,58.505,-51.139,-179.647,6.347,149.048
C06246=1150.981,58.754,-51.155,-179.644,6.349,149.048
C06247=1150.975,59.004,-51.171,-179.642,6.350,149.048
C06248=1150.971,59.253,-51.187,-179.639,6.351,149.047
C06249=1150.965,59.503,-51.203,-179.636,6.352,149.046
C06250=1150.961,59.752,-51.220,-179.634,6.354,149.046
C06251=1150.956,60.001,-51.235,-179.630,6.355,149.045
C06252=1150.951,60.251,-51.252,-179.628,6.356,149.045
C06253=1150.946,60.500,-51.268,-179.625,6.357,149.044
C06254=1150.940,60.750,-51.285,-179.623,6.358,149.044
C06255=1150.935,60.999,-51.300,-179.620,6.360,149.043
C06256=1150.930,61.248,-51.317,-179.618,6.360,149.043
C06257=1150.925,61.498,-51.333,-179.615,6.362,149.042
C06258=1150.920,61.747,-51.349,-179.613,6.363,149.042
C06259=1150.916,61.997,-51.366,-179.609,6.364,149.041
C06260=1150.910,62.246,-51.381,-179.607,6.365,149.041
C06261=1150.906,62.496,-51.398,-179.604,6.366,149.040
C06262=1150.900,62.745,-51.413,-179.602,6.367,149.040
C06263=1150.896,62.994,-51.430,-179.599,6.369,149.039
C06264=1150.891,63.244,-51.447,-179.596,6.370,149.039
C06265=1150.885,63.494,-51.463,-179.594,6.371,149.038
C06266=1150.881,63.743,-51.480,-179.591,6.372,149.038
C06267=1150.876,63.992,-51.496,-179.588,6.373,149.037
C06268=1150.871,64.242,-51.512,-179.586,6.375,149.037
C06269=1150.866,64.491,-51.528,-179.583,6.375,149.036
C06270=1150.861,64.740,-51.545,-179.580,6.377,149.035
C06271=1150.856,64.990,-51.561,-179.578,6.378,149.035
C06272=1150.851,65.239,-51.578,-179.575,6.379,149.035
C06273=1150.846,65.488,-51.594,-179.572,6.381,149.034
C06274=1150.841,65.738,-51.610,-179.570,6.381,149.033
C06275=1150.836,65.988,-51.627,-179.567,6.383,149.033
C06276=1150.831,66.237,-51.643,-179.565,6.384,149.032
C06277=1150.827,66.486,-51.660,-179.562,6.385,149.032
C06278=1150.821,66.736,-51.676,-179.559,6.386,149.031
C06279=1150.816,66.985,-51.693,-179.556,6.387,149.031
C06280=1150.812,67.235,-51.709,-179.554,6.389,149.030
C06281=1150.807,67.484,-51.725,-179.551,6.390,149.030
C06282=1150.801,67.734,-51.742,-179.548,6.391,149.029
C06283=1150.796,67.983,-51.758,-179.546,6.392,149.029
C06284=1150.792,68.232,-51.775,-179.543,6.393,149.028
C06285=1150.787,68.482,-51.792,-179.540,6.395,149.028
C06286=1150.781,68.731,-51.809,-179.538,6.396,149.027
C06287=1150.777,68.980,-51.825,-179.535,6.397,149.027
C06288=1150.771,69.230,-51.841,-179.533,6.398,149.026
C06289=1150.767,69.479,-51.858,-179.530,6.400,149.026
C06290=1150.762,69.729,-51.875,-179.527,6.401,149.025
C06291=1150.757,69.978,-51.891,-179.525,6.402,149.025
C06292=1150.752,70.227,-51.908,-179.522,6.404,149.024
C06293=1150.747,70.477,-51.925,-179.519,6.404,149.024
C06294=1150.742,70.726,-51.941,-179.516,6.406,149.023
C06295=1150.737,70.975,-51.958,-179.513,6.407,149.023
C06296=1150.732,71.225,-51.975,-179.511,6.408,149.022
C06297=1150.727,71.474,-51.992,-179.508,6.410,149.022
C06298=1150.723,71.723,-52.008,-179.506,6.410,149.021
C06299=1150.717,71.973,-52.025,-179.503,6.412,149.021
C06300=1150.712,72.222,-52.042,-179.500,6.413,149.020
C06301=1150.708,72.472,-52.058,-179.498,6.414,149.020
C06302=1150.702,72.722,-52.075,-179.495,6.416,149.019
C06303=1150.698,72.970,-52.092,-179.493,6.416,149.019
C06304=1150.692,73.220,-52.109,-179.489,6.418,149.018
C06305=1150.688,73.469,-52.126,-179.487,6.419,149.018
C06306=1150.683,73.718,-52.142,-179.485,6.420,149.017
C06307=1150.678,73.968,-52.160,-179.482,6.422,149.017
C06308=1150.673,74.217,-52.176,-179.479,6.423,149.016
C06309=1150.668,74.467,-52.193,-179.476,6.424,149.016
C06310=1150.663,74.716,-52.210,-179.474,6.426,149.015
C06311=1150.658,74.966,-52.227,-179.471,6.426,149.015
C06312=1150.653,75.215,-52.244,-179.468,6.428,149.014
C06313=1150.649,75.465,-52.260,-179.466,6.430,149.014
C06314=1150.643,75.714,-52.277,-179.463,6.430,149.013
C06315=1150.638,75.963,-52.294,-179.460,6.432,149.013
C06316=1150.633,76.213,-52.311,-179.458,6.433,149.012
C06317=1150.629,76.462,-52.329,-179.455,6.434,149.012
C06318=1150.623,76.711,-52.345,-179.452,6.436,149.011
C06319=1150.619,76.960,-52.362,-179.449,6.437,149.011
C06320=1150.613,77.210,-52.379,-179.447,6.438,149.010
C06321=1150.609,77.460,-52.396,-179.444,6.439,149.010
C06322=1150.603,77.708,-52.414,-179.441,6.441,149.009
C06323=1150.599,77.958,-52.430,-179.439,6.442,149.008
C06324=1150.594,78.208,-52.448,-179.436,6.443,149.008
C06325=1150.589,78.457,-52.464,-179.433,6.445,149.008
C06326=1150.584,78.707,-52.482,-179.431,6.445,149.007
C06327=1150.579,78.955,-52.499,-179.428,6.447,149.007
C06328=1150.574,79.205,-52.516,-179.426,6.448,149.006
C06329=1150.569,79.474,-52.535,-179.422,6.449,149.005
C06330=1150.563,79.741,-52.552,-179.420,6.451,149.005
C06331=1150.558,80.010,-52.571,-179.417,6.452,149.004
C06332=1150.553,80.279,-52.590,-179.414,6.454,149.004
C06333=1150.548,80.528,-52.607,-179.411,6.456,149.004
C06334=1150.543,80.777,-52.624,-179.408,6.456,149.003
C06335=1150.538,81.027,-52.641,-179.406,6.458,149.002
C06336=1150.533,81.276,-52.659,-179.403,6.460,149.002
C06337=1150.528,81.526,-52.676,-179.400,6.460,149.001
C06338=1150.524,81.775,-52.693,-179.398,6.462,149.001
C06339=1150.519,82.024,-52.711,-179.395,6.463,149.001
C06340=1150.513,82.274,-52.728,-179.393,6.464,149.000
C06341=1150.509,82.522,-52.745,-179.389,6.466,148.999
C06342=1150.503,82.772,-52.762,-179.387,6.467,148.999
C06343=1150.498,83.021,-52.780,-179.385,6.468,148.999
C06344=1150.494,83.271,-52.797,-179.381,6.469,148.998
C06345=1150.489,83.521,-52.814,-179.379,6.471,148.998
C06346=1150.484,83.770,-52.832,-179.376,6.473,148.997
C06347=1150.479,84.019,-52.849,-179.374,6.474,148.997
C06348=1150.474,84.268,-52.867,-179.371,6.475,148.996
C06349=1150.469,84.518,-52.884,-179.368,6.477,148.996
C06350=1150.464,84.766,-52.901,-179.366,6.477,148.995
C06351=1150.459,85.016,-52.918,-179.362,6.479,148.995
C06352=1150.454,85.265,-52.936,-179.360,6.480,148.994
C06353=1150.449,85.515,-52.953,-179.357,6.482,148.994
C06354=1150.445,85.764,-52.971,-179.355,6.483,148.993
C06355=1150.440,86.014,-52.988,-179.352,6.484,148.993
C06356=1150.435,86.263,-53.006,-179.349,6.486,148.992
C06357=1150.430,86.513,-53.023,-179.347,6.487,148.992
C06358=1150.425,86.762,-53.041,-179.344,6.488,148.991
C06359=1150.421,87.011,-53.059,-179.341,6.490,148.991
C06360=1150.415,87.261,-53.076,-179.338,6.492,148.990
C06361=1150.410,87.510,-53.094,-179.336,6.492,148.990
C06362=1150.405,87.760,-53.111,-179.333,6.494,148.989
C06363=1150.401,88.008,-53.129,-179.330,6.495,148.989
C06364=1150.396,88.258,-53.147,-179.328,6.496,148.988
C06365=1150.391,88.507,-53.164,-179.325,6.498,148.988
C06366=1150.386,88.757,-53.182,-179.322,6.499,148.987
C06367=1150.381,89.006,-53.199,-179.319,6.501,148.987
C06368=1150.376,89.256,-53.217,-179.317,6.502,148.986
C06369=1150.372,89.504,-53.234,-179.314,6.504,148.986
C06370=1150.367,89.754,-53.252,-179.311,6.505,148.985
C06371=1150.362,90.003,-53.270,-179.308,6.507,148.985
C06372=1150.357,90.253,-53.288,-179.306,6.507,148.985
C06373=1150.352,90.502,-53.306,-179.303,6.509,148.984
C06374=1150.346,90.751,-53.323,-179.300,6.510,148.983
C06375=1150.342,91.001,-53.341,-179.297,6.512,148.983
C06376=1150.337,91.250,-53.359,-179.295,6.513,148.983
C06377=1150.332,91.499,-53.376,-179.293,6.515,148.982
C06378=1150.327,91.749,-53.393,-179.289,6.516,148.982
C06379=1150.322,91.998,-53.411,-179.287,6.518,148.981
C06380=1150.317,92.247,-53.429,-179.284,6.518,148.981
C06381=1150.313,92.496,-53.447,-179.282,6.520,148.980
C06382=1150.308,92.745,-53.465,-179.279,6.521,148.980
C06383=1150.302,92.995,-53.483,-179.276,6.523,148.979
C06384=1150.298,93.244,-53.501,-179.274,6.524,148.979
C06385=1150.293,93.493,-53.519,-179.271,6.526,148.978
C06386=1150.288,93.743,-53.537,-179.268,6.527,148.978
C06387=1150.283,93.992,-53.555,-179.265,6.529,148.977
C06388=1150.278,94.242,-53.573,-179.263,6.530,148.977
C06389=1150.274,94.491,-53.591,-179.260,6.531,148.976
C06390=1150.269,94.740,-53.609,-179.257,6.533,148.976
C06391=1150.263,94.990,-53.626,-179.254,6.534,148.975
C06392=1150.259,95.239,-53.644,-179.251,6.536,148.975
C06393=1150.254,95.488,-53.662,-179.249,6.537,148.975
C06394=1150.249,95.737,-53.680,-179.246,6.538,148.974
C06395=1150.244,95.986,-53.698,-179.243,6.540,148.974
C06396=1150.239,96.236,-53.716,-179.241,6.542,148.973
C06397=1150.235,96.485,-53.734,-179.238,6.543,148.973
C06398=1150.230,96.735,-53.752,-179.235,6.544,148.972
C06399=1150.225,96.984,-53.770,-179.233,6.545,148.972
C06400=1150.220,97.233,-53.788,-179.230,6.547,148.971
C06401=1150.215,97.482,-53.806,-179.227,6.549,148.971
C06402=1150.210,97.731,-53.824,-179.225,6.550,148.970
C06403=1150.204,97.981,-53.843,-179.222,6.551,148.970
C06404=1150.200,98.231,-53.861,-179.219,6.553,148.969
C06405=1150.195,98.480,-53.879,-179.216,6.554,148.969
C06406=1150.190,98.729,-53.897,-179.214,6.556,148.968
C06407=1150.185,98.978,-53.915,-179.211,6.557,148.968
C06408=1150.180,99.227,-53.933,-179.208,6.558,148.967
C06409=1150.176,99.477,-53.952,-179.205,6.560,148.967
C06410=1150.171,99.726,-53.970,-179.203,6.562,148.967
C06411=1150.166,99.975,-53.989,-179.200,6.563,148.966
C06412=1150.161,100.225,-54.007,-179.197,6.565,148.966
C06413=1150.156,100.474,-54.025,-179.195,6.566,148.965
C06414=1150.152,100.724,-54.043,-179.192,6.567,148.965
C06415=1150.147,100.973,-54.061,-179.189,6.569,148.964
C06416=1150.142,101.221,-54.080,-179.186,6.571,148.964
C06417=1150.137,101.471,-54.098,-179.183,6.572,148.963
C06418=1150.132,101.720,-54.116,-179.181,6.573,148.963
C06419=1150.127,101.970,-54.135,-179.178,6.575,148.962
C06420=1150.122,102.219,-54.153,-179.176,6.576,148.962
C06421=1150.118,102.468,-54.171,-179.173,6.578,148.962
C06422=1150.112,102.717,-54.190,-179.170,6.579,148.961
C06423=1150.108,102.967,-54.208,-179.167,6.581,148.961
C06424=1150.103,103.216,-54.226,-179.165,6.582,148.960
C06425=1150.098,103.465,-54.245,-179.162,6.583,148.960
C06426=1150.093,103.714,-54.263,-179.159,6.585,148.959
C06427=1150.088,103.964,-54.282,-179.156,6.586,148.959
C06428=1150.083,104.213,-54.300,-179.153,6.588,148.958
C06429=1150.078,104.462,-54.319,-179.151,6.590,148.958
C06430=1150.074,104.712,-54.337,-179.148,6.592,148.957
C06431=1150.069,104.961,-54.355,-179.146,6.592,148.957
C06432=1150.064,105.210,-54.374,-179.143,6.594,148.957
C06433=1150.058,105.478,-54.394,-179.140,6.595,148.956
C06434=1150.054,105.747,-54.414,-179.137,6.597,148.956
C06435=1150.048,106.015,-54.435,-179.134,6.598,148.955
C06436=1150.043,106.283,-54.454,-179.131,6.601,148.955
C06437=1150.038,106.533,-54.473,-179.129,6.602,148.954
C06438=1150.034,106.782,-54.492,-179.126,6.604,148.954
C06439=1150.029,107.031,-54.510,-179.123,6.605,148.953
C06440=1150.023,107.281,-54.528,-179.120,6.607,148.953
C06441=1150.019,107.530,-54.547,-179.117,6.608,148.952
C06442=1150.013,107.780,-54.566,-179.114,6.610,148.952
C06443=1150.009,108.028,-54.585,-179.112,6.612,148.951
C06444=1150.005,108.278,-54.603,-179.109,6.613,148.951
C06445=1149.999,108.527,-54.622,-179.107,6.614,148.951
C06446=1149.994,108.776,-54.640,-179.104,6.616,148.950
C06447=1149.990,109.026,-54.660,-179.101,6.617,148.950
C06448=1149.985,109.275,-54.678,-179.098,6.619,148.949
C06449=1149.981,109.524,-54.697,-179.095,6.621,148.949
C06450=1149.975,109.774,-54.715,-179.093,6.622,148.948
C06451=1149.970,110.022,-54.734,-179.090,6.624,148.948
C06452=1149.965,110.272,-54.753,-179.087,6.625,148.947
C06453=1149.961,110.521,-54.772,-179.085,6.626,148.947
C06454=1149.956,110.770,-54.791,-179.082,6.628,148.946
C06455=1149.951,111.020,-54.809,-179.079,6.630,148.946
C06456=1149.946,111.268,-54.829,-179.076,6.631,148.946
C06457=1149.941,111.518,-54.847,-179.074,6.633,148.945
C06458=1149.936,111.767,-54.866,-179.071,6.635,148.945
C06459=1149.932,112.016,-54.885,-179.068,6.636,148.944
C06460=1149.926,112.266,-54.904,-179.065,6.638,148.944
C06461=1149.922,112.514,-54.923,-179.062,6.639,148.943
C06462=1149.917,112.764,-54.942,-179.060,6.641,148.943
C06463=1149.912,113.013,-54.960,-179.057,6.643,148.943
C06464=1149.907,113.263,-54.980,-179.055,6.644,148.942
C06465=1149.903,113.511,-54.999,-179.052,6.645,148.942
C06466=1149.898,113.762,-55.018,-179.049,6.647,148.941
C06467=1149.893,114.010,-55.036,-179.046,6.648,148.941
C06468=1149.888,114.260,-55.056,-179.043,6.650,148.940
C06469=1149.883,114.509,-55.075,-179.041,6.652,148.940
C06470=1149.879,114.758,-55.094,-179.038,6.654,148.940
C06471=1149.873,115.007,-55.113,-179.035,6.655,148.939
C06472=1149.869,115.256,-55.132,-179.033,6.657,148.939
C06473=1149.864,115.505,-55.151,-179.030,6.659,148.938
C06474=1149.858,115.755,-55.170,-179.027,6.660,148.938
C06475=1149.854,116.004,-55.189,-179.024,6.662,148.937
C06476=1149.849,116.253,-55.208,-179.021,6.663,148.937
C06477=1149.844,116.503,-55.228,-179.019,6.664,148.936
C06478=1149.840,116.752,-55.247,-179.016,6.666,148.936
C06479=1149.835,117.001,-55.266,-179.014,6.668,148.936
C06480=1149.830,117.251,-55.285,-179.011,6.669,148.935
C06481=1149.825,117.499,-55.304,-179.008,6.671,148.935
C06482=1149.821,117.749,-55.323,-179.005,6.672,148.934
C06483=1149.815,117.998,-55.343,-179.002,6.674,148.934
C06484=1149.811,118.247,-55.362,-179.000,6.676,148.933
C06485=1149.806,118.496,-55.381,-178.997,6.678,148.933
C06486=1149.801,118.746,-55.401,-178.994,6.679,148.933
C06487=1149.797,118.994,-55.419,-178.991,6.681,148.932
C06488=1149.792,119.244,-55.439,-178.989,6.683,148.932
C06489=1149.786,119.493,-55.458,-178.986,6.684,148.931
C06490=1149.782,119.742,-55.478,-178.983,6.686,148.931
C06491=1149.778,119.991,-55.497,-178.980,6.688,148.931
C06492=1149.772,120.240,-55.516,-178.977,6.689,148.930
C06493=1149.768,120.490,-55.536,-178.975,6.691,148.930
C06494=1149.762,120.739,-55.555,-178.972,6.692,148.929
C06495=1149.758,120.988,-55.574,-178.969,6.694,148.929
C06496=1149.754,121.238,-55.594,-178.966,6.696,148.928
C06497=1149.748,121.486,-55.613,-178.964,6.698,148.928
C06498=1149.743,121.736,-55.633,-178.961,6.699,148.928
C06499=1149.739,121.984,-55.652,-178.958,6.701,148.927
C06500=1149.734,122.234,-55.671,-178.955,6.703,148.927
C06501=1149.729,122.484,-55.691,-178.953,6.704,148.926
C06502=1149.724,122.733,-55.710,-178.951,6.705,148.926
C06503=1149.719,122.982,-55.730,-178.947,6.707,148.925
C06504=1149.715,123.232,-55.750,-178.945,6.708,148.925
C06505=1149.710,123.480,-55.769,-178.942,6.710,148.925
C06506=1149.705,123.729,-55.789,-178.939,6.712,148.924
C06507=1149.701,123.979,-55.808,-178.937,6.713,148.924
C06508=1149.695,124.228,-55.828,-178.934,6.715,148.923
C06509=1149.691,124.477,-55.847,-178.931,6.717,148.923
C06510=1149.686,124.727,-55.867,-178.928,6.719,148.923
C06511=1149.681,124.975,-55.887,-178.926,6.720,148.922
C06512=1149.676,125.225,-55.907,-178.923,6.722,148.922
C06513=1149.672,125.474,-55.926,-178.920,6.724,148.921
C06514=1149.667,125.723,-55.945,-178.918,6.725,148.921
C06515=1149.662,125.972,-55.965,-178.915,6.727,148.921
C06516=1149.658,126.221,-55.985,-178.912,6.729,148.920
C06517=1149.653,126.471,-56.005,-178.909,6.730,148.920
C06518=1149.647,126.720,-56.024,-178.906,6.732,148.919
C06519=1149.643,126.969,-56.044,-178.903,6.734,148.919
C06520=1149.638,127.218,-56.064,-178.900,6.736,148.918
C06521=1149.633,127.467,-56.083,-178.897,6.738,148.918
C06522=1149.629,127.716,-56.104,-178.895,6.739,148.918
C06523=1149.624,127.966,-56.123,-178.892,6.741,148.917
C06524=1149.619,128.215,-56.143,-178.889,6.743,148.917
C06525=1149.614,128.463,-56.163,-178.887,6.745,148.916
C06526=1149.609,128.713,-56.183,-178.884,6.746,148.916
C06527=1149.605,128.962,-56.202,-178.881,6.748,148.916
C06528=1149.600,129.211,-56.223,-178.878,6.750,148.915
C06529=1149.595,129.460,-56.242,-178.876,6.751,148.915
C06530=1149.590,129.709,-56.262,-178.873,6.753,148.914
C06531=1149.586,129.959,-56.282,-178.870,6.755,148.914
C06532=1149.581,130.208,-56.302,-178.868,6.757,148.914
C06533=1149.576,130.457,-56.322,-178.865,6.758,148.913
C06534=1149.571,130.706,-56.341,-178.862,6.760,148.913
C06535=1149.567,130.955,-56.362,-178.859,6.762,148.912
C06536=1149.562,131.205,-56.381,-178.857,6.763,148.912
C06537=1149.557,131.473,-56.404,-178.854,6.765,148.911
C06538=1149.552,131.742,-56.425,-178.850,6.767,148.911
C06539=1149.546,132.011,-56.446,-178.847,6.769,148.911
C06540=1149.541,132.279,-56.468,-178.845,6.771,148.910
C06541=1149.537,132.528,-56.488,-178.842,6.772,148.910
C06542=1149.532,132.776,-56.508,-178.839,6.774,148.909
C06543=1149.526,133.026,-56.528,-178.837,6.776,148.909
C06544=1149.522,133.275,-56.549,-178.834,6.778,148.909
C06545=1149.517,133.525,-56.568,-178.831,6.780,148.908
C06546=1149.512,133.774,-56.589,-178.828,6.782,148.908
C06547=1149.508,134.023,-56.609,-178.825,6.783,148.907
C06548=1149.503,134.272,-56.628,-178.822,6.785,148.907
C06549=1149.497,134.521,-56.649,-178.820,6.787,148.907
C06550=1149.493,134.770,-56.669,-178.817,6.789,148.906
C06551=1149.488,135.019,-56.689,-178.814,6.790,148.906
C06552=1149.484,135.268,-56.710,-178.812,6.792,148.906
C06553=1149.479,135.518,-56.729,-178.809,6.794,148.905
C06554=1149.474,135.767,-56.750,-178.806,6.795,148.905
C06555=1149.470,136.016,-56.771,-178.803,6.797,148.904
C06556=1149.464,136.264,-56.791,-178.801,6.799,148.904
C06557=1149.460,136.514,-56.810,-178.798,6.801,148.904
C06558=1149.455,136.763,-56.831,-178.795,6.803,148.903
C06559=1149.450,137.012,-56.852,-178.792,6.805,148.903
C06560=1149.445,137.262,-56.871,-178.789,6.807,148.902
C06561=1149.441,137.511,-56.892,-178.787,6.808,148.902
C06562=1149.436,137.760,-56.913,-178.784,6.810,148.902
C06563=1149.431,138.009,-56.933,-178.781,6.812,148.901
C06564=1149.427,138.258,-56.953,-178.778,6.813,148.901
C06565=1149.421,138.508,-56.974,-178.776,6.815,148.900
C06566=1149.417,138.757,-56.994,-178.773,6.817,148.900
C06567=1149.413,139.006,-57.014,-178.770,6.819,148.900
C06568=1149.408,139.255,-57.035,-178.767,6.821,148.899
C06569=1149.403,139.504,-57.056,-178.764,6.823,148.899
C06570=1149.398,139.753,-57.076,-178.762,6.824,148.899
C06571=1149.394,140.002,-57.096,-178.759,6.826,148.898
C06572=1149.389,140.252,-57.117,-178.756,6.828,148.898
C06573=1149.384,140.501,-57.137,-178.753,6.830,148.897
C06574=1149.379,140.750,-57.158,-178.751,6.831,148.897
C06575=1149.375,140.999,-57.178,-178.748,6.833,148.897
C06576=1149.370,141.248,-57.199,-178.745,6.835,148.896
C06577=1149.365,141.497,-57.220,-178.742,6.837,148.896
C06578=1149.360,141.746,-57.240,-178.739,6.839,148.895
C06579=1149.355,141.995,-57.261,-178.737,6.841,148.895
C06580=1149.351,142.244,-57.281,-178.734,6.842,148.895
C06581=1149.346,142.493,-57.302,-178.731,6.844,148.894
C06582=1149.341,142.742,-57.323,-178.728,6.846,148.894
C06583=1149.337,142.991,-57.343,-178.726,6.848,148.894
C06584=1149.332,143.241,-57.364,-178.723,6.850,148.893
C06585=1149.327,143.490,-57.384,-178.720,6.852,148.893
C06586=1149.322,143.739,-57.405,-178.718,6.854,148.893
C06587=1149.318,143.988,-57.426,-178.715,6.856,148.892
C06588=1149.312,144.237,-57.447,-178.712,6.857,148.892
C06589=1149.308,144.486,-57.467,-178.709,6.859,148.891
C06590=1149.304,144.735,-57.488,-178.707,6.861,148.891
C06591=1149.298,144.984,-57.508,-178.703,6.863,148.891
C06592=1149.294,145.233,-57.530,-178.701,6.865,148.890
C06593=1149.289,145.482,-57.551,-178.698,6.867,148.890
C06594=1149.284,145.731,-57.571,-178.695,6.868,148.889
C06595=1149.280,145.981,-57.592,-178.693,6.870,148.889
C06596=1149.275,146.230,-57.613,-178.690,6.872,148.889
C06597=1149.270,146.479,-57.634,-178.687,6.874,148.888
C06598=1149.266,146.727,-57.655,-178.684,6.876,148.888
C06599=1149.261,146.976,-57.676,-178.682,6.878,148.888
C06600=1149.256,147.226,-57.697,-178.679,6.880,148.887
C06601=1149.251,147.475,-57.718,-178.676,6.882,148.887
C06602=1149.246,147.724,-57.738,-178.673,6.883,148.887
C06603=1149.241,147.973,-57.760,-178.670,6.886,148.886
C06604=1149.238,148.222,-57.780,-178.667,6.888,148.886
C06605=1149.232,148.471,-57.801,-178.665,6.889,148.885
C06606=1149.227,148.721,-57.822,-178.662,6.891,148.885
C06607=1149.223,148.969,-57.843,-178.659,6.893,148.885
C06608=1149.218,149.218,-57.864,-178.657,6.894,148.884
C06609=1149.214,149.467,-57.885,-178.653,6.897,148.884
C06610=1149.209,149.716,-57.906,-178.651,6.899,148.884
C06611=1149.204,149.966,-57.928,-178.648,6.901,148.883
C06612=1149.200,150.215,-57.948,-178.646,6.903,148.883
C06613=1149.195,150.463,-57.970,-178.643,6.904,148.883
C06614=1149.190,150.713,-57.991,-178.640,6.907,148.882
C06615=1149.184,150.962,-58.012,-178.637,6.909,148.882
C06616=1149.181,151.211,-58.033,-178.634,6.910,148.882
C06617=1149.176,151.460,-58.054,-178.632,6.912,148.881
C06618=1149.171,151.709,-58.076,-178.629,6.914,148.881
C06619=1149.166,151.958,-58.096,-178.626,6.917,148.881
C06620=1149.162,152.206,-58.118,-178.623,6.918,148.880
C06621=1149.157,152.456,-58.139,-178.621,6.920,148.880
C06622=1149.152,152.706,-58.160,-178.618,6.922,148.879
C06623=1149.148,152.954,-58.181,-178.615,6.923,148.879
C06624=1149.143,153.203,-58.202,-178.612,6.926,148.879
C06625=1149.138,153.452,-58.224,-178.609,6.928,148.878
C06626=1149.133,153.702,-58.245,-178.607,6.929,148.878
C06627=1149.128,153.951,-58.267,-178.604,6.932,148.878
C06628=1149.124,154.199,-58.287,-178.601,6.934,148.877
C06629=1149.119,154.448,-58.309,-178.598,6.936,148.877
C06630=1149.115,154.697,-58.331,-178.596,6.938,148.877
C06631=1149.109,154.947,-58.352,-178.593,6.939,148.876
C06632=1149.105,155.195,-58.374,-178.590,6.941,148.876
C06633=1149.101,155.445,-58.394,-178.587,6.943,148.876
C06634=1149.096,155.694,-58.416,-178.585,6.946,148.875
C06635=1149.091,155.942,-58.438,-178.582,6.947,148.875
C06636=1149.086,156.192,-58.459,-178.579,6.949,148.875
C06637=1149.082,156.441,-58.481,-178.576,6.952,148.874
C06638=1149.076,156.690,-58.502,-178.573,6.953,148.874
C06639=1149.072,156.939,-58.523,-178.571,6.955,148.874
C06640=1149.067,157.188,-58.545,-178.568,6.957,148.873
C06641=1149.063,157.457,-58.568,-178.565,6.959,148.873
C06642=1149.057,157.727,-58.592,-178.562,6.961,148.872
C06643=1149.052,157.994,-58.615,-178.559,6.964,148.872
C06644=1149.046,158.264,-58.638,-178.556,6.965,148.872
C06645=1149.042,158.513,-58.660,-178.553,6.968,148.872
C06646=1149.038,158.761,-58.681,-178.550,6.970,148.871
C06647=1149.033,159.011,-58.702,-178.548,6.972,148.871
C06648=1149.029,159.260,-58.724,-178.545,6.973,148.870
C06649=1149.024,159.509,-58.746,-178.542,6.976,148.870
C06650=1149.020,159.758,-58.768,-178.539,6.978,148.870
C06651=1149.014,160.007,-58.789,-178.537,6.980,148.870
C06652=1149.009,160.256,-58.811,-178.534,6.981,148.869
C06653=1149.005,160.505,-58.833,-178.531,6.984,148.869
C06654=1149.000,160.754,-58.854,-178.528,6.986,148.868
C06655=1148.996,161.003,-58.876,-178.525,6.987,148.868
C06656=1148.991,161.252,-58.898,-178.523,6.990,148.868
C06657=1148.986,161.500,-58.920,-178.520,6.992,148.868
C06658=1148.982,161.750,-58.941,-178.517,6.994,148.867
C06659=1148.977,161.999,-58.963,-178.514,6.995,148.867
C06660=1148.973,162.248,-58.985,-178.511,6.998,148.866
C06661=1148.968,162.497,-59.007,-178.509,7.000,148.866
C06662=1148.962,162.746,-59.029,-178.506,7.002,148.866
C06663=1148.958,162.995,-59.051,-178.503,7.004,148.866
C06664=1148.953,163.244,-59.073,-178.500,7.006,148.865
C06665=1148.949,163.493,-59.095,-178.497,7.008,148.865
C06666=1148.944,163.742,-59.116,-178.495,7.010,148.865
C06667=1148.940,163.991,-59.138,-178.492,7.012,148.864
C06668=1148.935,164.240,-59.160,-178.489,7.014,148.864
C06669=1148.930,164.489,-59.182,-178.487,7.016,148.864
C06670=1148.926,164.738,-59.204,-178.483,7.018,148.863
C06671=1148.921,164.987,-59.226,-178.481,7.021,148.863
C06672=1148.916,165.236,-59.248,-178.478,7.022,148.863
C06673=1148.911,165.485,-59.270,-178.475,7.025,148.862
C06674=1148.907,165.734,-59.292,-178.472,7.027,148.862
C06675=1148.902,165.983,-59.314,-178.470,7.029,148.862
C06676=1148.898,166.231,-59.336,-178.467,7.031,148.861
C06677=1148.893,166.481,-59.358,-178.464,7.033,148.861
C06678=1148.888,166.730,-59.381,-178.461,7.035,148.861
C06679=1148.884,166.979,-59.403,-178.459,7.036,148.860
C06680=1148.879,167.228,-59.424,-178.456,7.039,148.860
C06681=1148.874,167.477,-59.446,-178.453,7.041,148.860
C06682=1148.870,167.726,-59.468,-178.451,7.043,148.859
C06683=1148.865,167.975,-59.491,-178.447,7.045,148.859
C06684=1148.860,168.223,-59.513,-178.445,7.047,148.859
C06685=1148.856,168.473,-59.535,-178.442,7.049,148.859
C06686=1148.851,168.721,-59.557,-178.439,7.052,148.858
C06687=1148.846,168.971,-59.579,-178.436,7.053,148.858
C06688=1148.841,169.219,-59.602,-178.434,7.055,148.858
C06689=1148.837,169.468,-59.624,-178.431,7.058,148.857
C06690=1148.832,169.718,-59.646,-178.428,7.060,148.857
C06691=1148.827,169.967,-59.668,-178.425,7.062,148.857
C06692=1148.823,170.215,-59.691,-178.423,7.064,148.856
C06693=1148.818,170.464,-59.713,-178.420,7.066,148.856
C06694=1148.813,170.714,-59.735,-178.417,7.069,148.856
C06695=1148.809,170.962,-59.758,-178.414,7.070,148.855
C06696=1148.804,171.211,-59.780,-178.412,7.072,148.855
C06697=1148.800,171.461,-59.802,-178.408,7.075,148.855
C06698=1148.795,171.709,-59.825,-178.406,7.077,148.854
C06699=1148.790,171.958,-59.847,-178.404,7.079,148.854
C06700=1148.786,172.207,-59.870,-178.400,7.081,148.854
C06701=1148.781,172.456,-59.892,-178.398,7.083,148.854
C06702=1148.776,172.705,-59.914,-178.395,7.085,148.853
C06703=1148.772,172.953,-59.937,-178.392,7.088,148.853
C06704=1148.767,173.203,-59.960,-178.389,7.089,148.853
C06705=1148.763,173.452,-59.982,-178.386,7.092,148.852
C06706=1148.758,173.700,-60.004,-178.384,7.094,148.852
C06707=1148.753,173.949,-60.027,-178.381,7.096,148.852
C06708=1148.749,174.199,-60.049,-178.378,7.098,148.852
C06709=1148.743,174.447,-60.072,-178.375,7.100,148.851
C06710=1148.739,174.696,-60.094,-178.373,7.102,148.851
C06711=1148.734,174.946,-60.118,-178.370,7.105,148.851
C06712=1148.730,175.194,-60.139,-178.367,7.106,148.850
C06713=1148.725,175.443,-60.163,-178.364,7.109,148.850
C06714=1148.721,175.693,-60.185,-178.361,7.111,148.850
C06715=1148.715,175.941,-60.208,-178.359,7.113,148.849
C06716=1148.711,176.190,-60.230,-178.356,7.116,148.849
C06717=1148.706,176.439,-60.253,-178.353,7.117,148.849
C06718=1148.702,176.688,-60.276,-178.350,7.120,148.849
C06719=1148.697,176.937,-60.298,-178.347,7.122,148.848
C06720=1148.693,177.186,-60.321,-178.345,7.124,148.848
C06721=1148.688,177.435,-60.344,-178.342,7.126,148.848
C06722=1148.684,177.684,-60.366,-178.339,7.128,148.847
C06723=1148.679,177.932,-60.389,-178.336,7.131,148.847
C06724=1148.674,178.182,-60.412,-178.334,7.133,148.847
C06725=1148.670,178.431,-60.435,-178.331,7.135,148.847
C06726=1148.666,178.679,-60.458,-178.328,7.137,148.846
C06727=1148.660,178.928,-60.481,-178.325,7.139,148.846
C06728=1148.655,179.177,-60.503,-178.322,7.142,148.846
C06729=1148.651,179.426,-60.526,-178.320,7.144,148.846
C06730=1148.647,179.675,-60.549,-178.317,7.146,148.845
C06731=1148.642,179.923,-60.572,-178.314,7.148,148.845
C06732=1148.637,180.173,-60.594,-178.312,7.150,148.845
C06733=1148.632,180.422,-60.618,-178.308,7.153,148.844
C06734=1148.628,180.671,-60.641,-178.306,7.154,148.844
C06735=1148.624,180.920,-60.664,-178.303,7.157,148.844
C06736=1148.618,181.168,-60.687,-178.300,7.159,148.844
C06737=1148.614,181.417,-60.709,-178.298,7.161,148.843
C06738=1148.609,181.666,-60.732,-178.295,7.164,148.843
C06739=1148.605,181.915,-60.756,-178.292,7.165,148.843
C06740=1148.601,182.164,-60.778,-178.289,7.168,148.843
C06741=1148.596,182.413,-60.802,-178.287,7.170,148.842
C06742=1148.591,182.661,-60.825,-178.283,7.173,148.842
C06743=1148.587,182.910,-60.848,-178.281,7.175,148.842
C06744=1148.582,183.159,-60.871,-178.278,7.177,148.841
C06745=1148.577,183.429,-60.896,-178.275,7.179,148.841
C06746=1148.572,183.699,-60.921,-178.272,7.182,148.841
C06747=1148.567,183.968,-60.945,-178.269,7.185,148.841
C06748=1148.562,184.239,-60.971,-178.266,7.186,148.840
C06749=1148.557,184.487,-60.994,-178.263,7.189,148.840
C06750=1148.552,184.736,-61.017,-178.261,7.191,148.840
C06751=1148.548,184.985,-61.040,-178.258,7.193,148.839
C06752=1148.544,185.234,-61.063,-178.255,7.196,148.839
C06753=1148.539,185.482,-61.087,-178.252,7.198,148.839
C06754=1148.534,185.731,-61.111,-178.249,7.200,148.839
C06755=1148.530,185.980,-61.134,-178.247,7.203,148.838
C06756=1148.526,186.229,-61.157,-178.244,7.205,148.838
C06757=1148.521,186.478,-61.180,-178.241,7.207,148.838
C06758=1148.516,186.727,-61.204,-178.238,7.209,148.838
C06759=1148.512,186.976,-61.227,-178.235,7.212,148.837
C06760=1148.506,187.224,-61.250,-178.233,7.214,148.837
C06761=1148.502,187.473,-61.273,-178.230,7.216,148.837
C06762=1148.497,187.722,-61.297,-178.227,7.218,148.837
C06763=1148.493,187.971,-61.320,-178.224,7.221,148.836
C06764=1148.489,188.220,-61.343,-178.221,7.223,148.836
C06765=1148.484,188.469,-61.367,-178.219,7.226,148.836
C06766=1148.479,188.718,-61.390,-178.216,7.227,148.835
C06767=1148.475,188.967,-61.414,-178.214,7.230,148.835
C06768=1148.470,189.215,-61.438,-178.210,7.232,148.835
C06769=1148.465,189.464,-61.461,-178.208,7.234,148.835
C06770=1148.461,189.713,-61.484,-178.205,7.237,148.835
C06771=1148.456,189.962,-61.508,-178.202,7.238,148.834
C06772=1148.452,190.211,-61.532,-178.199,7.241,148.834
C06773=1148.447,190.460,-61.555,-178.197,7.243,148.834
C06774=1148.442,190.709,-61.579,-178.194,7.246,148.834
C06775=1148.438,190.958,-61.602,-178.191,7.248,148.833
C06776=1148.433,191.206,-61.626,-178.188,7.251,148.833
C06777=1148.428,191.455,-61.649,-178.185,7.253,148.833
C06778=1148.424,191.704,-61.673,-178.182,7.255,148.832
C06779=1148.419,191.953,-61.697,-178.180,7.258,148.832
C06780=1148.415,192.202,-61.720,-178.177,7.260,148.832
C06781=1148.410,192.450,-61.744,-178.174,7.263,148.832
C06782=1148.406,192.699,-61.768,-178.171,7.264,148.831
C06783=1148.401,192.948,-61.791,-178.169,7.267,148.831
C06784=1148.396,193.197,-61.815,-178.166,7.269,148.831
C06785=1148.392,193.446,-61.838,-178.163,7.272,148.831
C06786=1148.387,193.694,-61.862,-178.160,7.274,148.831
C06787=1148.383,193.944,-61.886,-178.158,7.276,148.830
C06788=1148.379,194.192,-61.910,-178.155,7.278,148.830
C06789=1148.373,194.441,-61.934,-178.152,7.281,148.830
C06790=1148.369,194.690,-61.958,-178.150,7.283,148.830
C06791=1148.364,194.939,-61.982,-178.147,7.286,148.829
C06792=1148.360,195.187,-62.006,-178.144,7.288,148.829
C06793=1148.355,195.436,-62.029,-178.141,7.290,148.829
C06794=1148.351,195.685,-62.053,-178.138,7.293,148.829
C06795=1148.346,195.934,-62.076,-178.135,7.295,148.828
C06796=1148.342,196.182,-62.101,-178.132,7.298,148.828
C06797=1148.337,196.432,-62.125,-178.130,7.299,148.828
C06798=1148.333,196.681,-62.149,-178.127,7.302,148.828
C06799=1148.328,196.929,-62.173,-178.124,7.304,148.827
C06800=1148.323,197.178,-62.196,-178.121,7.307,148.827
C06801=1148.319,197.427,-62.220,-178.119,7.309,148.827
C06802=1148.314,197.676,-62.244,-178.116,7.312,148.827
C06803=1148.309,197.924,-62.268,-178.113,7.313,148.826
C06804=1148.305,198.173,-62.293,-178.110,7.316,148.826
C06805=1148.301,198.422,-62.316,-178.107,7.319,148.826
C06806=1148.296,198.671,-62.340,-178.105,7.321,148.826
C06807=1148.291,198.920,-62.365,-178.102,7.324,148.826
C06808=1148.287,199.168,-62.389,-178.100,7.326,148.825
C06809=1148.283,199.418,-62.413,-178.097,7.329,148.825
C06810=1148.278,199.666,-62.437,-178.094,7.330,148.825
C06811=1148.273,199.915,-62.462,-178.091,7.333,148.825
C06812=1148.269,200.163,-62.486,-178.088,7.336,148.825
C06813=1148.264,200.412,-62.509,-178.086,7.338,148.824
C06814=1148.260,200.662,-62.534,-178.082,7.340,148.824
C06815=1148.255,200.910,-62.558,-178.080,7.343,148.824
C06816=1148.251,201.159,-62.582,-178.077,7.345,148.824
C06817=1148.246,201.407,-62.607,-178.074,7.348,148.824
C06818=1148.241,201.656,-62.630,-178.072,7.350,148.823
C06819=1148.237,201.905,-62.655,-178.069,7.353,148.823
C06820=1148.232,202.154,-62.679,-178.066,7.354,148.823
C06821=1148.228,202.403,-62.703,-178.063,7.357,148.823
C06822=1148.224,202.652,-62.728,-178.060,7.360,148.823
C06823=1148.219,202.900,-62.752,-178.058,7.362,148.822
C06824=1148.214,203.149,-62.777,-178.055,7.365,148.822
C06825=1148.210,203.397,-62.801,-178.052,7.367,148.822
C06826=1148.205,203.647,-62.826,-178.049,7.370,148.822
C06827=1148.201,203.895,-62.850,-178.046,7.372,148.821
C06828=1148.196,204.144,-62.874,-178.044,7.374,148.821
C06829=1148.191,204.392,-62.898,-178.041,7.377,148.821
C06830=1148.187,204.642,-62.924,-178.039,7.379,148.821
C06831=1148.183,204.890,-62.948,-178.036,7.382,148.821
C06832=1148.177,205.139,-62.972,-178.032,7.384,148.820
C06833=1148.174,205.388,-62.997,-178.030,7.386,148.820
C06834=1148.169,205.636,-63.021,-178.027,7.389,148.820
C06835=1148.164,205.885,-63.045,-178.025,7.391,148.820
C06836=1148.160,206.134,-63.070,-178.021,7.394,148.819
C06837=1148.155,206.383,-63.095,-178.019,7.397,148.819
C06838=1148.151,206.631,-63.119,-178.016,7.399,148.819
C06839=1148.146,206.881,-63.144,-178.013,7.401,148.819
C06840=1148.141,207.129,-63.168,-178.010,7.404,148.819
C06841=1148.137,207.378,-63.192,-178.008,7.406,148.818
C06842=1148.132,207.627,-63.218,-178.005,7.409,148.818
C06843=1148.128,207.875,-63.242,-178.002,7.412,148.818
C06844=1148.123,208.124,-63.267,-177.999,7.414,148.818
C06845=1148.119,208.373,-63.291,-177.997,7.416,148.818
C06846=1148.114,208.622,-63.316,-177.994,7.418,148.817
C06847=1148.110,208.871,-63.340,-177.991,7.421,148.817
C06848=1148.105,209.119,-63.366,-177.988,7.424,148.817
C06849=1148.100,209.389,-63.393,-177.985,7.427,148.817
C06850=1148.096,209.660,-63.420,-177.982,7.430,148.817
C06851=1148.091,209.931,-63.447,-177.979,7.432,148.816
C06852=1148.086,210.201,-63.473,-177.976,7.435,148.816
C06853=1148.081,210.450,-63.498,-177.974,7.437,148.816
C06854=1148.076,210.699,-63.523,-177.971,7.440,148.816
C06855=1148.072,210.947,-63.548,-177.968,7.443,148.816
C06856=1148.068,211.196,-63.573,-177.965,7.444,148.815
C06857=1148.063,211.445,-63.598,-177.962,7.447,148.815
C06858=1148.059,211.693,-63.623,-177.960,7.450,148.815
C06859=1148.054,211.942,-63.647,-177.957,7.452,148.815
C06860=1148.049,212.192,-63.672,-177.954,7.455,148.815
C06861=1148.045,212.440,-63.698,-177.951,7.457,148.815
C06862=1148.040,212.688,-63.722,-177.949,7.460,148.814
C06863=1148.036,212.937,-63.748,-177.946,7.462,148.814
C06864=1148.031,213.186,-63.772,-177.943,7.465,148.814
C06865=1148.027,213.435,-63.797,-177.940,7.467,148.814
C06866=1148.022,213.683,-63.822,-177.938,7.470,148.814
C06867=1148.018,213.932,-63.847,-177.934,7.473,148.813
C06868=1148.013,214.180,-63.873,-177.932,7.475,148.813
C06869=1148.009,214.430,-63.897,-177.929,7.478,148.813
C06870=1148.004,214.678,-63.922,-177.926,7.480,148.813
C06871=1148.000,214.927,-63.947,-177.923,7.483,148.813
C06872=1147.995,215.175,-63.973,-177.921,7.485,148.813
C06873=1147.990,215.425,-63.998,-177.918,7.488,148.812
C06874=1147.987,215.673,-64.023,-177.915,7.491,148.812
C06875=1147.982,215.921,-64.048,-177.913,7.493,148.812
C06876=1147.978,216.171,-64.073,-177.910,7.495,148.812
C06877=1147.973,216.419,-64.099,-177.907,7.498,148.812
C06878=1147.968,216.668,-64.124,-177.905,7.500,148.812
C06879=1147.963,216.916,-64.149,-177.902,7.503,148.812
C06880=1147.960,217.165,-64.174,-177.899,7.506,148.811
C06881=1147.955,217.413,-64.199,-177.896,7.509,148.811
C06882=1147.951,217.662,-64.225,-177.894,7.511,148.811
C06883=1147.946,217.911,-64.251,-177.890,7.513,148.811
C06884=1147.941,218.160,-64.275,-177.887,7.516,148.811
C06885=1147.937,218.409,-64.301,-177.885,7.518,148.810
C06886=1147.932,218.657,-64.326,-177.882,7.521,148.810
C06887=1147.928,218.906,-64.351,-177.879,7.524,148.810
C06888=1147.923,219.155,-64.377,-177.876,7.527,148.810
C06889=1147.919,219.403,-64.403,-177.874,7.529,148.810
C06890=1147.914,219.652,-64.428,-177.871,7.532,148.810
C06891=1147.911,219.900,-64.453,-177.868,7.534,148.809
C06892=1147.906,220.149,-64.478,-177.865,7.537,148.809
C06893=1147.901,220.398,-64.504,-177.863,7.539,148.809
C06894=1147.897,220.646,-64.529,-177.860,7.542,148.809
C06895=1147.892,220.895,-64.555,-177.857,7.545,148.809
C06896=1147.888,221.144,-64.581,-177.854,7.548,148.809
C06897=1147.883,221.392,-64.606,-177.852,7.550,148.808
C06898=1147.879,221.641,-64.631,-177.849,7.553,148.808
C06899=1147.875,221.890,-64.657,-177.846,7.556,148.808
C06900=1147.870,222.138,-64.682,-177.843,7.558,148.808
C06901=1147.866,222.387,-64.708,-177.841,7.560,148.808
C06902=1147.861,222.636,-64.734,-177.838,7.563,148.808
C06903=1147.856,222.884,-64.760,-177.835,7.566,148.808
C06904=1147.852,223.133,-64.786,-177.832,7.569,148.808
C06905=1147.847,223.382,-64.811,-177.830,7.571,148.807
C06906=1147.843,223.630,-64.837,-177.827,7.574,148.807
C06907=1147.838,223.879,-64.862,-177.824,7.577,148.807
C06908=1147.834,224.127,-64.888,-177.821,7.579,148.807
C06909=1147.830,224.376,-64.914,-177.818,7.581,148.807
C06910=1147.825,224.624,-64.939,-177.816,7.584,148.806
C06911=1147.821,224.873,-64.965,-177.813,7.587,148.806
C06912=1147.816,225.122,-64.991,-177.810,7.590,148.806
C06913=1147.812,225.371,-65.017,-177.808,7.592,148.806
C06914=1147.807,225.619,-65.043,-177.805,7.595,148.806
C06915=1147.803,225.868,-65.068,-177.802,7.598,148.806
C06916=1147.798,226.117,-65.094,-177.799,7.601,148.806
C06917=1147.794,226.365,-65.120,-177.796,7.603,148.806
C06918=1147.789,226.613,-65.147,-177.794,7.605,148.805
C06919=1147.785,226.862,-65.172,-177.791,7.608,148.805
C06920=1147.780,227.111,-65.198,-177.788,7.611,148.805
C06921=1147.776,227.360,-65.224,-177.785,7.614,148.805
C06922=1147.772,227.609,-65.250,-177.782,7.617,148.805
C06923=1147.766,227.857,-65.276,-177.780,7.619,148.805
C06924=1147.762,228.105,-65.302,-177.777,7.622,148.805
C06925=1147.758,228.354,-65.328,-177.774,7.624,148.804
C06926=1147.754,228.603,-65.353,-177.771,7.627,148.804
C06927=1147.749,228.852,-65.380,-177.769,7.630,148.804
C06928=1147.745,229.099,-65.406,-177.766,7.632,148.804
C06929=1147.740,229.348,-65.432,-177.763,7.635,148.804
C06930=1147.736,229.597,-65.457,-177.760,7.638,148.804
C06931=1147.731,229.846,-65.484,-177.758,7.641,148.804
C06932=1147.727,230.094,-65.510,-177.755,7.644,148.804
C06933=1147.723,230.343,-65.536,-177.752,7.646,148.803
C06934=1147.717,230.591,-65.562,-177.749,7.648,148.803
C06935=1147.713,230.840,-65.588,-177.746,7.651,148.803
C06936=1147.709,231.088,-65.614,-177.744,7.654,148.803
C06937=1147.705,231.337,-65.641,-177.741,7.657,148.803
C06938=1147.700,231.586,-65.667,-177.738,7.660,148.803
C06939=1147.695,231.835,-65.693,-177.735,7.662,148.803
C06940=1147.691,232.083,-65.720,-177.733,7.665,148.802
C06941=1147.687,232.332,-65.746,-177.730,7.668,148.802
C06942=1147.682,232.580,-65.772,-177.727,7.671,148.802
C06943=1147.678,232.828,-65.798,-177.724,7.674,148.802
C06944=1147.673,233.077,-65.825,-177.721,7.677,148.802
C06945=1147.669,233.326,-65.851,-177.719,7.678,148.802
C06946=1147.665,233.574,-65.877,-177.716,7.681,148.802
C06947=1147.660,233.823,-65.904,-177.713,7.684,148.802
C06948=1147.656,234.071,-65.930,-177.710,7.687,148.802
C06949=1147.651,234.320,-65.956,-177.708,7.690,148.801
C06950=1147.647,234.569,-65.983,-177.705,7.693,148.801
C06951=1147.642,234.818,-66.009,-177.703,7.695,148.801
C06952=1147.638,235.066,-66.036,-177.699,7.698,148.801
C06953=1147.633,235.338,-66.064,-177.697,7.701,148.801
C06954=1147.629,235.609,-66.093,-177.693,7.704,148.801
C06955=1147.623,235.881,-66.122,-177.690,7.707,148.801
C06956=1147.618,236.153,-66.151,-177.688,7.710,148.801
C06957=1147.614,236.401,-66.178,-177.684,7.713,148.800
C06958=1147.609,236.650,-66.205,-177.682,7.716,148.800
C06959=1147.605,236.899,-66.230,-177.679,7.719,148.800
C06960=1147.600,237.147,-66.257,-177.676,7.721,148.800
C06961=1147.597,237.395,-66.284,-177.674,7.724,148.800
C06962=1147.592,237.644,-66.311,-177.671,7.727,148.800
C06963=1147.587,237.893,-66.337,-177.668,7.729,148.800
C06964=1147.583,238.141,-66.364,-177.665,7.732,148.800
C06965=1147.578,238.390,-66.391,-177.662,7.735,148.799
C06966=1147.574,238.638,-66.417,-177.659,7.738,148.799
C06967=1147.570,238.888,-66.444,-177.657,7.741,148.799
C06968=1147.565,239.136,-66.471,-177.654,7.744,148.799
C06969=1147.562,239.384,-66.498,-177.652,7.746,148.799
C06970=1147.557,239.633,-66.525,-177.649,7.749,148.799
C06971=1147.552,239.881,-66.552,-177.646,7.752,148.799
C06972=1147.548,240.130,-66.577,-177.643,7.755,148.799
C06973=1147.543,240.379,-66.604,-177.640,7.758,148.799
C06974=1147.539,240.627,-66.632,-177.638,7.760,148.799
C06975=1147.535,240.875,-66.658,-177.635,7.763,148.799
C06976=1147.530,241.124,-66.685,-177.632,7.766,148.798
C06977=1147.525,241.372,-66.712,-177.629,7.769,148.798
C06978=1147.522,241.620,-66.739,-177.627,7.771,148.798
C06979=1147.517,241.869,-66.766,-177.624,7.774,148.798
C06980=1147.512,242.117,-66.793,-177.621,7.777,148.798
C06981=1147.509,242.366,-66.820,-177.618,7.780,148.798
C06982=1147.504,242.615,-66.847,-177.616,7.783,148.798
C06983=1147.500,242.863,-66.874,-177.613,7.786,148.798
C06984=1147.495,243.112,-66.901,-177.610,7.789,148.798
C06985=1147.490,243.360,-66.928,-177.607,7.791,148.798
C06986=1147.486,243.608,-66.954,-177.604,7.794,148.798
C06987=1147.482,243.857,-66.981,-177.602,7.797,148.798
C06988=1147.477,244.105,-67.008,-177.599,7.799,148.797
C06989=1147.473,244.355,-67.036,-177.597,7.802,148.797
C06990=1147.469,244.603,-67.062,-177.594,7.805,148.797
C06991=1147.464,244.851,-67.089,-177.591,7.808,148.797
C06992=1147.460,245.100,-67.116,-177.588,7.811,148.797
C06993=1147.455,245.348,-67.143,-177.585,7.814,148.797
C06994=1147.451,245.596,-67.171,-177.583,7.817,148.797
C06995=1147.447,245.845,-67.199,-177.579,7.820,148.797
C06996=1147.442,246.094,-67.226,-177.577,7.823,148.797
C06997=1147.438,246.342,-67.252,-177.574,7.825,148.797
C06998=1147.433,246.591,-67.279,-177.571,7.828,148.796
C06999=1147.429,246.839,-67.306,-177.568,7.831,148.796
C07000=1147.425,247.088,-67.334,-177.565,7.834,148.796
C07001=1147.420,247.336,-67.362,-177.563,7.836,148.796
C07002=1147.416,247.585,-67.389,-177.560,7.839,148.796
C07003=1147.411,247.833,-67.416,-177.558,7.842,148.796
C07004=1147.407,248.082,-67.444,-177.555,7.845,148.796
C07005=1147.403,248.330,-67.471,-177.552,7.848,148.796
C07006=1147.398,248.579,-67.498,-177.549,7.851,148.796
C07007=1147.394,248.827,-67.526,-177.547,7.854,148.796
C07008=1147.389,249.075,-67.553,-177.544,7.857,148.796
C07009=1147.385,249.324,-67.580,-177.541,7.860,148.796
C07010=1147.381,249.572,-67.608,-177.538,7.863,148.796
C07011=1147.376,249.821,-67.635,-177.535,7.866,148.795
C07012=1147.372,250.070,-67.662,-177.533,7.869,148.795
C07013=1147.368,250.318,-67.690,-177.530,7.871,148.795
C07014=1147.363,250.566,-67.717,-177.527,7.874,148.795
C07015=1147.359,250.814,-67.745,-177.524,7.877,148.795
C07016=1147.354,251.063,-67.772,-177.521,7.880,148.795
C07017=1147.350,251.311,-67.800,-177.519,7.883,148.795
C07018=1147.345,251.560,-67.827,-177.516,7.886,148.795
C07019=1147.342,251.808,-67.855,-177.513,7.889,148.795
C07020=1147.337,252.057,-67.883,-177.510,7.892,148.795
C07021=1147.333,252.305,-67.910,-177.508,7.895,148.795
C07022=1147.329,252.554,-67.938,-177.506,7.897,148.795
C07023=1147.324,252.802,-67.966,-177.503,7.900,148.795
C07024=1147.320,253.050,-67.993,-177.500,7.903,148.795
C07025=1147.315,253.299,-68.021,-177.497,7.906,148.795
C07026=1147.310,253.548,-68.048,-177.495,7.909,148.795
C07027=1147.306,253.795,-68.076,-177.492,7.912,148.795
C07028=1147.302,254.045,-68.104,-177.489,7.915,148.794
C07029=1147.298,254.292,-68.131,-177.486,7.918,148.794
C07030=1147.293,254.540,-68.159,-177.484,7.921,148.794
C07031=1147.289,254.790,-68.187,-177.481,7.924,148.794
C07032=1147.284,255.038,-68.215,-177.478,7.927,148.794
C07033=1147.280,255.286,-68.243,-177.475,7.930,148.794
C07034=1147.276,255.535,-68.270,-177.472,7.932,148.794
C07035=1147.271,255.783,-68.298,-177.470,7.935,148.794
C07036=1147.268,256.031,-68.326,-177.467,7.938,148.794
C07037=1147.262,256.280,-68.354,-177.464,7.941,148.794
C07038=1147.259,256.529,-68.382,-177.462,7.945,148.794
C07039=1147.254,256.777,-68.410,-177.459,7.947,148.794
C07040=1147.250,257.024,-68.437,-177.456,7.950,148.794
C07041=1147.245,257.273,-68.466,-177.453,7.953,148.794
C07042=1147.241,257.522,-68.493,-177.451,7.956,148.794
C07043=1147.237,257.770,-68.521,-177.448,7.959,148.794
C07044=1147.232,258.019,-68.550,-177.445,7.962,148.794
C07045=1147.228,258.267,-68.578,-177.442,7.965,148.794
C07046=1147.224,258.515,-68.606,-177.439,7.968,148.794
C07047=1147.220,258.764,-68.633,-177.437,7.971,148.793
C07048=1147.215,259.012,-68.661,-177.434,7.974,148.793
C07049=1147.211,259.261,-68.690,-177.432,7.977,148.794
C07050=1147.207,259.509,-68.717,-177.429,7.980,148.793
C07051=1147.202,259.758,-68.746,-177.426,7.983,148.793
C07052=1147.198,260.006,-68.774,-177.423,7.986,148.793
C07053=1147.193,260.255,-68.803,-177.420,7.989,148.793
C07054=1147.189,260.502,-68.830,-177.418,7.992,148.793
C07055=1147.185,260.751,-68.859,-177.415,7.995,148.793
C07056=1147.180,260.999,-68.887,-177.412,7.998,148.793
C07057=1147.175,261.272,-68.918,-177.409,8.001,148.793
C07058=1147.171,261.546,-68.948,-177.406,8.004,148.793
C07059=1147.166,261.820,-68.980,-177.403,8.008,148.793
C07060=1147.162,262.093,-69.011,-177.400,8.011,148.793
C07061=1147.156,262.341,-69.040,-177.397,8.014,148.793
C07062=1147.153,262.590,-69.068,-177.395,8.017,148.793
C07063=1147.148,262.837,-69.096,-177.392,8.020,148.793
C07064=1147.144,263.086,-69.124,-177.389,8.023,148.793
C07065=1147.140,263.334,-69.152,-177.386,8.026,148.793
C07066=1147.135,263.583,-69.181,-177.384,8.029,148.793
C07067=1147.131,263.832,-69.209,-177.381,8.032,148.793
C07068=1147.126,264.080,-69.237,-177.378,8.035,148.793
C07069=1147.123,264.328,-69.266,-177.376,8.038,148.793
C07070=1147.118,264.576,-69.295,-177.373,8.041,148.793
C07071=1147.114,264.825,-69.323,-177.370,8.045,148.793
C07072=1147.109,265.074,-69.351,-177.367,8.048,148.793
C07073=1147.104,265.322,-69.380,-177.364,8.051,148.793
C07074=1147.101,265.570,-69.409,-177.362,8.054,148.793
C07075=1147.096,265.818,-69.437,-177.359,8.057,148.793
C07076=1147.092,266.066,-69.465,-177.356,8.060,148.793
C07077=1147.088,266.315,-69.494,-177.353,8.063,148.793
C07078=1147.084,266.563,-69.522,-177.351,8.066,148.793
C07079=1147.079,266.811,-69.551,-177.348,8.069,148.793
C07080=1147.074,267.060,-69.580,-177.345,8.072,148.793
C07081=1147.071,267.308,-69.608,-177.343,8.075,148.793
C07082=1147.066,267.556,-69.637,-177.340,8.078,148.793
C07083=1147.061,267.805,-69.666,-177.338,8.081,148.793
C07084=1147.057,268.053,-69.694,-177.335,8.084,148.793
C07085=1147.053,268.302,-69.723,-177.332,8.087,148.793
C07086=1147.048,268.550,-69.751,-177.329,8.090,148.793
C07087=1147.044,268.798,-69.780,-177.326,8.093,148.792
C07088=1147.040,269.047,-69.809,-177.323,8.097,148.793
C07089=1147.036,269.295,-69.839,-177.321,8.100,148.793
C07090=1147.031,269.543,-69.866,-177.318,8.103,148.793
C07091=1147.027,269.791,-69.896,-177.315,8.106,148.792
C07092=1147.023,270.040,-69.925,-177.313,8.109,148.793
C07093=1147.018,270.287,-69.954,-177.310,8.112,148.793
C07094=1147.014,270.536,-69.982,-177.307,8.115,148.793
C07095=1147.010,270.784,-70.011,-177.304,8.118,148.792
C07096=1147.006,271.033,-70.040,-177.302,8.121,148.792
C07097=1147.002,271.280,-70.068,-177.299,8.124,148.793
C07098=1146.997,271.529,-70.097,-177.297,8.127,148.793
C07099=1146.993,271.778,-70.127,-177.293,8.130,148.792
C07100=1146.989,272.026,-70.156,-177.290,8.133,148.792
C07101=1146.984,272.274,-70.184,-177.288,8.137,148.793
C07102=1146.980,272.522,-70.213,-177.285,8.140,148.793
C07103=1146.976,272.771,-70.242,-177.283,8.143,148.792
C07104=1146.971,273.019,-70.271,-177.280,8.146,148.793
C07105=1146.967,273.267,-70.301,-177.277,8.149,148.793
C07106=1146.962,273.516,-70.329,-177.275,8.152,148.793
C07107=1146.958,273.764,-70.359,-177.272,8.155,148.792
C07108=1146.955,274.012,-70.388,-177.270,8.158,148.793
C07109=1146.950,274.261,-70.416,-177.266,8.162,148.793
C07110=1146.945,274.508,-70.445,-177.263,8.165,148.793
C07111=1146.941,274.757,-70.475,-177.261,8.168,148.793
C07112=1146.937,275.005,-70.504,-177.258,8.171,148.793
C07113=1146.932,275.254,-70.533,-177.256,8.174,148.793
C07114=1146.928,275.502,-70.563,-177.253,8.177,148.793
C07115=1146.924,275.750,-70.592,-177.250,8.180,148.793
C07116=1146.919,275.998,-70.621,-177.248,8.183,148.793
C07117=1146.915,276.246,-70.651,-177.245,8.186,148.793
C07118=1146.912,276.494,-70.679,-177.242,8.190,148.793
C07119=1146.907,276.743,-70.708,-177.239,8.193,148.793
C07120=1146.903,276.991,-70.738,-177.236,8.196,148.793
C07121=1146.899,277.239,-70.767,-177.234,8.199,148.793
C07122=1146.895,277.488,-70.797,-177.231,8.202,148.793
C07123=1146.890,277.736,-70.826,-177.229,8.205,148.793
C07124=1146.886,277.984,-70.855,-177.226,8.208,148.793
C07125=1146.882,278.232,-70.884,-177.223,8.211,148.793
C07126=1146.877,278.480,-70.914,-177.220,8.215,148.793
C07127=1146.873,278.728,-70.943,-177.217,8.218,148.793
C07128=1146.869,278.977,-70.973,-177.215,8.221,148.793
C07129=1146.865,279.225,-71.002,-177.212,8.224,148.793
C07130=1146.861,279.473,-71.032,-177.210,8.227,148.793
C07131=1146.856,279.721,-71.061,-177.207,8.230,148.793
C07132=1146.852,279.970,-71.091,-177.204,8.233,148.793
C07133=1146.847,280.218,-71.121,-177.201,8.237,148.793
C07134=1146.843,280.467,-71.150,-177.199,8.240,148.793
C07135=1146.839,280.715,-71.180,-177.196,8.243,148.793
C07136=1146.835,280.963,-71.209,-177.193,8.246,148.793
C07137=1146.830,281.211,-71.238,-177.191,8.249,148.793
C07138=1146.826,281.459,-71.268,-177.188,8.252,148.793
C07139=1146.822,281.707,-71.297,-177.186,8.255,148.793
C07140=1146.818,281.955,-71.327,-177.182,8.259,148.793
C07141=1146.813,282.203,-71.357,-177.180,8.262,148.794
C07142=1146.809,282.452,-71.387,-177.177,8.265,148.793
C07143=1146.804,282.700,-71.416,-177.174,8.268,148.793
C07144=1146.800,282.948,-71.446,-177.172,8.272,148.794
C07145=1146.796,283.196,-71.475,-177.169,8.275,148.794
C07146=1146.792,283.444,-71.506,-177.166,8.279,148.794
C07147=1146.787,283.693,-71.535,-177.164,8.282,148.794
C07148=1146.783,283.941,-71.565,-177.161,8.285,148.794
C07149=1146.779,284.189,-71.594,-177.158,8.288,148.794
C07150=1146.775,284.437,-71.624,-177.156,8.291,148.794
C07151=1146.770,284.685,-71.654,-177.153,8.294,148.794
C07152=1146.766,284.934,-71.684,-177.150,8.298,148.794
C07153=1146.762,285.181,-71.714,-177.147,8.301,148.794
C07154=1146.757,285.430,-71.744,-177.145,8.304,148.794
C07155=1146.754,285.679,-71.774,-177.142,8.307,148.794
C07156=1146.750,285.927,-71.804,-177.140,8.310,148.794
C07157=1146.746,286.175,-71.834,-177.136,8.314,148.794
C07158=1146.741,286.423,-71.864,-177.134,8.317,148.794
C07159=1146.737,286.671,-71.894,-177.131,8.320,148.794
C07160=1146.733,286.919,-71.923,-177.129,8.323,148.794
C07161=1146.727,287.194,-71.957,-177.126,8.327,148.794
C07162=1146.723,287.470,-71.991,-177.123,8.330,148.794
C07163=1146.718,287.745,-72.023,-177.120,8.334,148.795
C07164=1146.714,288.020,-72.057,-177.117,8.338,148.795
C07165=1146.709,288.269,-72.087,-177.114,8.341,148.795
C07166=1146.705,288.517,-72.117,-177.112,8.344,148.795
C07167=1146.701,288.765,-72.147,-177.109,8.347,148.795
C07168=1146.697,289.013,-72.178,-177.106,8.350,148.795
C07169=1146.692,289.261,-72.207,-177.103,8.354,148.795
C07170=1146.688,289.509,-72.238,-177.101,8.357,148.795
C07171=1146.684,289.757,-72.268,-177.098,8.360,148.795
C07172=1146.680,290.006,-72.298,-177.096,8.364,148.795
C07173=1146.676,290.254,-72.329,-177.093,8.366,148.795
C07174=1146.672,290.502,-72.358,-177.090,8.371,148.795
C07175=1146.667,290.750,-72.389,-177.087,8.374,148.795
C07176=1146.663,290.998,-72.419,-177.085,8.377,148.795
C07177=1146.658,291.246,-72.449,-177.082,8.380,148.795
C07178=1146.655,291.495,-72.479,-177.079,8.384,148.796
C07179=1146.650,291.743,-72.510,-177.076,8.387,148.796
C07180=1146.646,291.990,-72.540,-177.074,8.390,148.796
C07181=1146.641,292.239,-72.570,-177.071,8.393,148.796
C07182=1146.638,292.487,-72.601,-177.069,8.396,148.796
C07183=1146.634,292.735,-72.632,-177.066,8.400,148.796
C07184=1146.630,292.983,-72.662,-177.063,8.403,148.796
C07185=1146.625,293.231,-72.692,-177.061,8.406,148.796
C07186=1146.621,293.479,-72.722,-177.058,8.409,148.796
C07187=1146.617,293.728,-72.753,-177.055,8.414,148.796
C07188=1146.612,293.976,-72.784,-177.052,8.416,148.796
C07189=1146.608,294.223,-72.814,-177.050,8.420,148.797
C07190=1146.603,294.472,-72.844,-177.047,8.423,148.797
C07191=1146.600,294.720,-72.875,-177.045,8.426,148.797
C07192=1146.596,294.968,-72.906,-177.042,8.430,148.797
C07193=1146.591,295.216,-72.936,-177.039,8.433,148.797
C07194=1146.587,295.464,-72.966,-177.037,8.436,148.797
C07195=1146.583,295.713,-72.998,-177.034,8.439,148.797
C07196=1146.579,295.960,-73.028,-177.031,8.443,148.797
C07197=1146.575,296.208,-73.059,-177.029,8.446,148.797
C07198=1146.571,296.457,-73.090,-177.026,8.449,148.797
C07199=1146.567,296.704,-73.120,-177.023,8.452,148.797
C07200=1146.562,296.952,-73.151,-177.021,8.456,148.798
C07201=1146.557,297.200,-73.181,-177.018,8.460,148.798
C07202=1146.554,297.449,-73.212,-177.015,8.463,148.798
C07203=1146.550,297.697,-73.243,-177.013,8.466,148.798
C07204=1146.545,297.945,-73.273,-177.010,8.470,148.798
C07205=1146.541,298.193,-73.305,-177.007,8.473,148.798
C07206=1146.537,298.441,-73.335,-177.005,8.476,148.798
C07207=1146.532,298.689,-73.366,-177.002,8.479,148.798
C07208=1146.528,298.938,-73.397,-176.999,8.483,148.798
C07209=1146.524,299.186,-73.427,-176.997,8.486,148.798
C07210=1146.520,299.433,-73.458,-176.994,8.489,148.799
C07211=1146.516,299.681,-73.489,-176.991,8.494,148.799
C07212=1146.512,299.929,-73.520,-176.989,8.496,148.799
C07213=1146.508,300.178,-73.551,-176.986,8.500,148.799
C07214=1146.503,300.426,-73.582,-176.984,8.503,148.799
C07215=1146.499,300.673,-73.612,-176.981,8.507,148.799
C07216=1146.495,300.921,-73.644,-176.978,8.510,148.799
C07217=1146.491,301.169,-73.675,-176.976,8.513,148.799
C07218=1146.487,301.418,-73.706,-176.973,8.516,148.799
C07219=1146.482,301.666,-73.737,-176.970,8.520,148.800
C07220=1146.478,301.913,-73.768,-176.968,8.523,148.800
C07221=1146.474,302.162,-73.799,-176.965,8.527,148.800
C07222=1146.470,302.410,-73.830,-176.962,8.531,148.800
C07223=1146.466,302.658,-73.861,-176.960,8.534,148.800
C07224=1146.462,302.906,-73.892,-176.957,8.537,148.800
C07225=1146.457,303.154,-73.923,-176.955,8.540,148.800
C07226=1146.453,303.402,-73.955,-176.951,8.544,148.800
C07227=1146.449,303.650,-73.986,-176.949,8.547,148.800
C07228=1146.445,303.898,-74.017,-176.947,8.550,148.801
C07229=1146.440,304.146,-74.048,-176.943,8.554,148.801
C07230=1146.436,304.394,-74.079,-176.941,8.557,148.801
C07231=1146.432,304.642,-74.111,-176.939,8.561,148.801
C07232=1146.428,304.890,-74.142,-176.936,8.565,148.801
C07233=1146.424,305.138,-74.173,-176.933,8.568,148.801
C07234=1146.420,305.386,-74.204,-176.931,8.571,148.801
C07235=1146.415,305.634,-74.235,-176.928,8.574,148.802
C07236=1146.411,305.882,-74.267,-176.925,8.578,148.802
C07237=1146.407,306.130,-74.298,-176.923,8.581,148.802
C07238=1146.403,306.378,-74.330,-176.920,8.585,148.802
C07239=1146.399,306.626,-74.360,-176.918,8.589,148.802
C07240=1146.395,306.874,-74.392,-176.915,8.592,148.802
C07241=1146.391,307.122,-74.424,-176.912,8.595,148.802
C07242=1146.387,307.370,-74.455,-176.910,8.599,148.803
C07243=1146.382,307.618,-74.486,-176.907,8.602,148.803
C07244=1146.378,307.866,-74.518,-176.904,8.605,148.803
C07245=1146.374,308.114,-74.549,-176.902,8.609,148.803
C07246=1146.369,308.362,-74.581,-176.899,8.612,148.803
C07247=1146.365,308.610,-74.612,-176.897,8.616,148.803
C07248=1146.361,308.858,-74.644,-176.894,8.620,148.803
C07249=1146.357,309.105,-74.676,-176.891,8.623,148.803
C07250=1146.353,309.354,-74.707,-176.889,8.626,148.804
C07251=1146.349,309.602,-74.738,-176.886,8.630,148.804
C07252=1146.345,309.849,-74.770,-176.883,8.633,148.804
C07253=1146.340,310.098,-74.802,-176.881,8.636,148.804
C07254=1146.336,310.346,-74.833,-176.878,8.640,148.804
C07255=1146.332,310.594,-74.865,-176.876,8.644,148.804
C07256=1146.328,310.842,-74.897,-176.873,8.647,148.805
C07257=1146.324,311.089,-74.928,-176.870,8.651,148.805
C07258=1146.320,311.337,-74.960,-176.868,8.654,148.805
C07259=1146.315,311.585,-74.992,-176.865,8.657,148.805
C07260=1146.311,311.833,-75.023,-176.862,8.661,148.805
C07261=1146.308,312.081,-75.055,-176.860,8.665,148.805
C07262=1146.303,312.329,-75.087,-176.857,8.668,148.805
C07263=1146.299,312.577,-75.119,-176.854,8.672,148.806
C07264=1146.295,312.825,-75.151,-176.852,8.675,148.806
C07265=1146.291,313.103,-75.187,-176.849,8.679,148.806
C07266=1146.285,313.381,-75.222,-176.846,8.683,148.806
C07267=1146.281,313.659,-75.258,-176.843,8.687,148.806
C07268=1146.276,313.935,-75.293,-176.840,8.691,148.806
C07269=1146.272,314.184,-75.325,-176.838,8.694,148.807
C07270=1146.268,314.432,-75.357,-176.835,8.697,148.807
C07271=1146.264,314.680,-75.389,-176.832,8.702,148.807
C07272=1146.260,314.927,-75.421,-176.830,8.705,148.807
C07273=1146.256,315.176,-75.453,-176.828,8.708,148.807
C07274=1146.252,315.424,-75.485,-176.824,8.712,148.807
C07275=1146.247,315.671,-75.517,-176.822,8.715,148.808
C07276=1146.243,315.919,-75.549,-176.819,8.719,148.808
C07277=1146.240,316.167,-75.581,-176.817,8.722,148.808
C07278=1146.235,316.415,-75.614,-176.814,8.726,148.808
C07279=1146.231,316.662,-75.645,-176.812,8.730,148.808
C07280=1146.227,316.910,-75.677,-176.809,8.733,148.809
C07281=1146.223,317.159,-75.710,-176.806,8.737,148.809
C07282=1146.219,317.407,-75.741,-176.804,8.740,148.809
C07283=1146.214,317.655,-75.773,-176.801,8.743,148.809
C07284=1146.211,317.902,-75.806,-176.798,8.747,148.809
C07285=1146.206,318.150,-75.838,-176.796,8.751,148.809
C07286=1146.203,318.398,-75.870,-176.794,8.754,148.810
C07287=1146.198,318.646,-75.902,-176.791,8.758,148.810
C07288=1146.194,318.893,-75.935,-176.788,8.761,148.810
C07289=1146.190,319.141,-75.967,-176.785,8.765,148.810
C07290=1146.186,319.390,-75.999,-176.783,8.769,148.810
C07291=1146.182,319.638,-76.031,-176.781,8.772,148.811
C07292=1146.178,319.886,-76.064,-176.778,8.776,148.811
C07293=1146.174,320.133,-76.096,-176.776,8.779,148.811
C07294=1146.169,320.381,-76.128,-176.773,8.783,148.811
C07295=1146.166,320.629,-76.161,-176.770,8.786,148.811
C07296=1146.161,320.877,-76.193,-176.768,8.790,148.812
C07297=1146.157,321.125,-76.226,-176.765,8.794,148.812
C07298=1146.154,321.373,-76.258,-176.762,8.797,148.812
C07299=1146.149,321.620,-76.290,-176.759,8.801,148.812
C07300=1146.145,321.868,-76.323,-176.757,8.804,148.812
C07301=1146.141,322.116,-76.355,-176.754,8.808,148.813
C07302=1146.137,322.364,-76.388,-176.752,8.812,148.813
C07303=1146.133,322.612,-76.420,-176.750,8.815,148.813
C07304=1146.129,322.860,-76.453,-176.747,8.819,148.813
C07305=1146.125,323.108,-76.485,-176.744,8.822,148.813
C07306=1146.121,323.355,-76.518,-176.741,8.826,148.814
C07307=1146.116,323.603,-76.550,-176.739,8.830,148.814
C07308=1146.112,323.851,-76.583,-176.737,8.833,148.814
C07309=1146.108,324.099,-76.615,-176.734,8.837,148.814
C07310=1146.105,324.346,-76.648,-176.731,8.840,148.814
C07311=1146.100,324.594,-76.681,-176.729,8.844,148.815
C07312=1146.096,324.842,-76.714,-176.726,8.848,148.815
C07313=1146.092,325.090,-76.747,-176.723,8.852,148.815
C07314=1146.088,325.338,-76.779,-176.721,8.855,148.815
C07315=1146.084,325.586,-76.812,-176.718,8.859,148.815
C07316=1146.080,325.834,-76.845,-176.716,8.862,148.816
C07317=1146.076,326.082,-76.877,-176.713,8.866,148.816
C07318=1146.072,326.329,-76.910,-176.710,8.870,148.816
C07319=1146.068,326.577,-76.943,-176.708,8.873,148.816
C07320=1146.063,326.825,-76.976,-176.705,8.877,148.817
C07321=1146.059,327.073,-77.009,-176.703,8.880,148.817
C07322=1146.056,327.321,-77.041,-176.700,8.884,148.817
C07323=1146.052,327.568,-77.074,-176.698,8.888,148.817
C07324=1146.047,327.817,-77.107,-176.695,8.892,148.818
C07325=1146.043,328.064,-77.140,-176.693,8.895,148.818
C07326=1146.039,328.312,-77.173,-176.691,8.898,148.818
C07327=1146.036,328.560,-77.206,-176.688,8.903,148.818
C07328=1146.032,328.807,-77.239,-176.685,8.906,148.818
C07329=1146.027,329.055,-77.272,-176.682,8.910,148.819
C07330=1146.023,329.303,-77.304,-176.680,8.913,148.819
C07331=1146.019,329.551,-77.338,-176.677,8.917,148.819
